FUNCTION "GCS7_BinCtrlSub" : VOID	// FC 67
TITLE = Bin Control: Subroutines
//COPYRIGHT:    (C) 1994 BY  BUHLER LTD.
//                           CH-9240 UZWIL  SWITZERLAND
//
//PRODUCT:      GCS7
//
//TITLE:        BIN CONTROL: SUBROUTINS
//
//-------------------------------------------------------------------------
//
//IDENT:        AUTOR:              DEPT:                         DATE:
//FC67.2.8      A.Egli              CT3                           18-Mai-2006
//                WinAC is not compatible
//FC67.2.7      A.Egli              CT3                           07-Jul-2004
//              DPFault per bin
//FC67.2.6      A.Egli              CT3                           08-Mar-2004
//              Per Bin bit InfIsInRecipe
//FC67.2.5      K.Tischer           CT3                           24-Oct-2003
//              - correction for StaLastBinActiv
//              - init test recipe 
//FC67.2.4      A.Egli              CT3                           04-Sep-2003
//              - check wit target value
//FC67.2.3      K.Tischer           CT3                           04-Jul-2003
//              - init DBW36 for decode
//FC67.2.2      A.Egli              CT3                           23-Jun-2003
//              - Set "BinDB".ToASW.BinActual also for Blend
//FC67.2.1      A.Egli              CT3                           05-Jun-2003
//              - Delete WeightTarget not before bin is deselected
//FC67.2.0      A.Egli              CT3                           07-Oct-2002
//              - New release 
//              - LastIngredient Active
//FC67.1.3      A.Egli              CT3                           06-Nov-01
//              subroutine 14: Init TestRefill
//FC67.1.2      A.Egli              AEE61                         14-Jan-98
//              Convert S5 to S7 (Version 1C)
//FC67.1.1      A.Egli              AEE61                         24-Jun-96
//              Convert S5 to S7 (Version 1C)
//
//-------------------------------------------------------------------------
//
//PURPOSE:      MANUAL : BINMAN
//
//RESTRICTIONS:
//
//-------------------------------------------------------------------------
//
//
//PARAMETER:
//------------
//  CODE: CODE OF CALLED FUNCTION
//        1  : Subroutine Test  Recipe
//        2  : Subroutine Read  Bin
//        3  : Subroutine Store Bin
//        4  : Subroutine Deselect All
//        5  : Subroutine Bin_Modify
//        6  : Subroutine Claer Value
//        7  : Subroutine Maske Active Bin
//        10 : Subroutine Read Ingredient
//        11 : Subroutine Read First Ingredient
//        12 : Subroutine Read Next Ingredient
//        13 : Subroutine Read_Blend_recipe
//
//ACTUAL DB BY CALL: DB Bin control
//AUFGESCHALGENER  : DB Siloverwaltung
//
//
AUTHOR : EA
FAMILY : GCS90UL
NAME : BIN_SUBR
VERSION : 2.8
VAR_INPUT
  CODE : INT ;	// CODE
END_VAR
VAR_TEMP
  BinNr : INT ;
  BinStatus : STRUCT
   InfLevelWarning : BOOL ;
   InfLevelFault1 : BOOL ;
   B10 : BOOL ;
   B11 : BOOL ;
   VarFlagOverwrite : BOOL ;
   InfLowLevel : BOOL ;
   InfLevelMiddle : BOOL ;
   InfHighLevel : BOOL ;
   InfActive : BOOL ;
   InfPreselect : BOOL ;
   InfDeselect : BOOL ;
   B3 : BOOL ;
   B4 : BOOL ;
   VarFlageLevelWarning : BOOL ;
   VarFlagLevelFault : BOOL ;
  END_STRUCT ;
  VarCntBin : INT ;
  VarAddrBin : DWORD ;
  VarCntIngr : INT ;
  VarAddrIngr : DINT ;
  VarBinNr : INT ;
  VarLenBinBit : INT ;	//Length of Bin data in bits
  VarLenIngrBit : INT ;	//Lenght per Ingr. in bits
  VarOkIngrCnt : INT ;	//Number of available ingredient (Transport)
  tmpNoTargetValue : BOOL ;
END_VAR
BEGIN
NETWORK
TITLE =
      L     DBW 10;	// "BinDB".Para.ParNoOfBytePerBin
      SLD   3;
      T     #VarLenBinBit;
      L     DBW 16;	// "BinDB".Para.ParNoOfBytePerIngr
      SLD   3;
      T     #VarLenIngrBit;
NETWORK
TITLE =  Subroutine Test Bin Status (Code=0)
//======================================
//
//Subroutine test bin Status: Code= 0
//-------------------------------------
//Input:
//Output:
//  DBX   43.0            // "BinDB".ToASW.InfActive
//  DBX   43.1            // "BinDB".ToASW.InfPreselect
//  DBX   43.2            // "BinDB".ToASW.InfDeselect 
//  DBX  103.0            // "BinDB".PCRead.Fault.EsLocked
//  DBX  103.1            // "BinDB".PCRead.Fault.EsLevelFault
//  DBX  105.7            // "BinDB".PCRead.Status.StaFeedOff
//  DBX   42.2            // "BinDB".ToASW.InfAllLocked
//  DBX   42.3            // "BinDB".ToASW.InfAllLevelFault
//
      L     #CODE;
      L     0;
      <>I;
      JC    aEnd;
      R     DBX 43.0;	// "BinDB".ToASW.InfActive
      R     DBX 43.1;	// "BinDB".ToASW.InfPreselect
      R     DBX 43.2;	// "BinDB".ToASW.InfDeselect 
      R     DBX 103.0;	// "BinDB".PCRead.Fault.EsLocked
      R     DBX 103.1;	// "BinDB".PCRead.Fault.EsLevelFault
      R     DBX 105.7;	// "BinDB".PCRead.Status.StaFeedOff
      R     DBX 104.3;	// "BinDB".PCRead.Status.StaDPFault     [2.7]
      S     DBX 42.2;	// "BinDB".ToASW.InfAllLocked
      S     DBX 42.3;	// "BinDB".ToASW.InfAllLevelFault
// [2.5] 
      S     DBX 43.4;	// "BinDB".ToASW.OutDryFillingDone
      L     0;
      T     DBW 56;	//"BinDB1".ToASW.OutActiveBinsCnt
      AN    DBX 7.0;	// ParObjectType=Blend
      JC    aAc1;
      T     DBW 48;	// "BinDB".ToASW.BinActual //[2.2]
//Start Adress Loop
aAc1: L     DBW 8;	//"BinDB".Para.ParByteFirstBin
      +     2;
      SLD   3;
      T     #VarAddrBin;	//--> Pointer to statusword of the bin
// (--loop bin: test  ----------)
      L     0;
      L     DBW 12;	//  "BinDB".Para.ParNoOfBin
      ==I;
      JC    aFER;
aLop: T     #VarCntBin;	// var_loop_bin_counter
      L     DBW [#VarAddrBin];	// binlist[n].Bin status word
      T     DBW 24;	//  )->var_bin_status
      AN    DBX 25.0;	//"BinDB".VarTemp.Bin.InfActiveBin
      JC    aEPY;
//Counter Active bins
      L     DBW 56;	//"BinDB1".ToASW.OutActiveBinsCnt
      +     1;
      T     DBW 56;	//"BinDB1".ToASW.OutActiveBinsCnt
      AN    DBX 7.0;	//[2.2 -->] ParObjectType=Blend
      JC    aAc2;
      L     #VarAddrBin;
      +     L#-16;
      LAR1;
      L     DBW [AR1,P#0.0];	// binlist[n].ParBinNr
      T     DBW 48;	// "BinDB".ToASW.BinActual     [<--2.2]
//Emptying Time
aAc2: LAR1  #VarAddrBin;
      L     DBW [AR1,P#2.0];	// binlist[n].ParEmptyingTime
      T     DBW 52;	// "BinDB".ToASW.OutEmptyingTimeBin
aEPY: A     DBX 25.0;	//"BinDB".VarTemp.Bin.InfActiveBin
      S     DBX 43.0;	// "BinDB".ToASW.InfActive
      A     DBX 25.1;	//"BinDB".VarTemp.Bin.InfPreselect
      S     DBX 43.1;	// "BinDB".ToASW.InfPreselect
      A     DBX 25.2;	// "BinDB".VarTemp.Bin.InfDeselect
      S     DBX 43.2;	//"BinDB".ToASW.InfDeselect
// --- DryFilling done ----------------
      A     DBX 25.0;	//"BinDB".VarTemp.Bin.InfActiveBin
      AN    DBX 24.3;	//"BinDB".VarTemp.Bin.OutDryFillingDone
      R     DBX 43.4;	// "BinDB".ToASW.OutDryFillingDone
// --- Feed Off ----------------
      A     DBX 25.0;	//"BinDB".VarTemp.Bin.InfActiveBin
      A     DBX 24.2;	//"BinDB".VarTemp.Bin.InFeedOff
      S     DBX 105.7;	// "BinDB".PCRead.Status.StaFeedOff
// --- DPFault ----------------
      A     DBX 25.0;	//"BinDB".VarTemp.Bin.InfActiveBin     [2.7]
      A     DBX 25.4;	//"BinDB".VarTemp.Bin.InOutDPFault     [2.7]
      S     DBX 104.3;	//"BinDB".PCRead.Status.StaDPFault     [2.7]
// --- Locked ----------------
      AN    DBX 24.0;	// bin[n]."BinDB".VarTemp.Bin.InfLocked
      JC    aR_W;
      A     DBX 25.0;	// "BinDB".VarTemp.Bin.InfActiveBin
      S     DBX 103.0;	// "BinDB".PCRead.Fault.EsLocked
      AN    DBX 25.6;	// "BinDB".VarTemp.Bin.VarFlagLocked
      S     DBX 25.6;	// "BinDB".VarTemp.Bin.VarFlagLocked
      S     DBX 41.0;	// "BinDB".ChangeBit.CBit1
      S     DBX 39.7;	// "BinDB".VarTemp.Value10.Flag7
      JU    aL_F;	// -- no warning --------------
aR_W: A     DBX 25.0;	// "BinDB".VarTemp.Bin.InfActiveBin
      R     DBX 42.2;	// "BinDB".ToASW.InfAllLocked
      A     DBX 25.6;	// "BinDB".VarTemp.Bin.VarFlagLocked
      R     DBX 25.6;	// "BinDB".VarTemp.Bin.VarFlagLocked 
      S     DBX 41.0;	// "BinDB".ChangeBit.CBit1
      S     DBX 39.7;	// "BinDB".VarTemp.Value10.Flag7
//---Faulted ----------------
aL_F: AN    DBX 24.1;	// "BinDB".VarTemp.Bin.InfLevelFault
      JC    aR_F;
//    --- fault ------------------
      A     DBX 25.0;	// "BinDB".VarTemp.Bin.InfActiveBin 
      S     DBX 103.1;	// "BinDB".PCRead.Fault.EsLevelFault
      AN    DBX 25.7;	// "BinDB".VarTemp.Bin.VarFlagLevelFault
      S     DBX 25.7;	// "BinDB".VarTemp.Bin.VarFlagLevelFault
      S     DBX 41.0;	// "BinDB".ChangeBit.CBit1 
      S     DBX 39.7;	// "BinDB".VarTemp.Value10.Flag7
      JU    aSAV;
//    -- no fault   --------------
aR_F: A     DBX 25.0;	//  "BinDB".VarTemp.Bin.InfActiveBin
      R     DBX 42.3;	//  "BinDB".ToASW.InfAllLevelFault 
      A     DBX 25.7;	//  "BinDB".VarTemp.Bin.VarFlagLevelFault
      R     DBX 25.7;	//  "BinDB".VarTemp.Bin.VarFlagLevelFault 
      S     DBX 41.0;	//  "BinDB".ChangeBit.CBit1 
      S     DBX 39.7;	// "BinDB".VarTemp.Value10.Flag7
//Store Bin
aSAV: L     DBW 24;	//   var_bin_status
      T     DBW [#VarAddrBin];	//   -> binlist[n].bin_status
      L     #VarAddrBin;
      L     #VarLenBinBit;
      +D;
      T     #VarAddrBin;	//   
      L     #VarCntBin;	//   
      LOOP  aLop;
//  (--END LOOP TEST -----------)
aFER: AN    DBX 43.0;	// "BinDB".ToASW.InfActive
      R     DBX 42.2;	// "BinDB".ToASW.InfAllLocked 
      R     DBX 42.3;	// "BinDB".ToASW.InfAllLevelFault 
      BEU;
aEnd: NOP   0;
NETWORK
TITLE = subroutine:Test recipe (Code 1)
//Input: DBW20="BinDB".VarTemp.InValue     = Source Recipe DBNr
//Input: DBW22="BinDB".VarTemp.BinNrByteNr = Source Recipe First Byte
//Output: DBW24=out.err_bin / BinStatus
//Output: DBW26=Number availabel ingredient 
//Output: DBW36=var_bin-number ingredient(error)
//Output: DBX39.1="BinDB".VarTemp.Value10.tmpLevelFault
//Output: DBX39.2="BinDB".VarTemp.Value10.tmpBinNotFound2
//Output: DBX39.3="BinDB".VarTemp.Value10.tmpEmptyRecipe
//Output: DBX39.4="BinDB".VarTemp.Value10.tmpFull
//Output: DBX39.6="BinDB".VarTemp.Value10.tmpLocked
//
      L     #CODE;
      L     1;
      <>I;
      JC    bEnd;
      S     DBX 39.6;	//"BinDB".VarTemp.Value10.tmpLocked
      S     DBX 39.1;	//"BinDB".VarTemp.Value10.tmpLevelFault
      S     DBX 39.4;	//"BinDB".VarTemp.Value10.tmpFull
      R     DBX 39.2;	//"BinDB".VarTemp.Value10.tmpBinNotFound2
      S     DBX 39.3;	//"BinDB".VarTemp.Value10.tmpEmptyRecipe
      L     0;	// [2.0]
      T     #VarOkIngrCnt;	// [2.0]
      T     DBW 36;	// [2.3]
// Init
      OPN   DI [DBW 20];	// Call Source DB: DBW20=inp.DB-Nr_source_recipe
      L     DBW 22;	// inp.ByteNrSourceRecipe
      +     6;	// Offset first ingredient
      SLD   3;	//   
      T     #VarAddrIngr;	//--> Address first ingredient
// ====START LOOP INGREDIENT =====
      L     0;
      L     DBW 18;	//  "BinDB".Para.ParNoOfIngr
      ==I;
      BEC;
bLoI: T     #VarCntIngr;
      L     DIW [#VarAddrIngr];	// load Ingredient bin number
      T     #VarBinNr;	// 
      L     0;	// 
      ==I;	// empty ingredient
      JC    bNXT;	// 
      L     DBW 8;	// "BinDB".Para.ParByteFirstBin
      SLD   3;	// 
      T     #VarAddrBin;	//--> Address of first bin
// ====START LOOP BIN ============
      L     1;
bLoB: T     #VarCntBin;	//   
      L     DBW 12;	// "BinDB".Para.ParNoOfBin 
      >I;
      JC    bErr;
      L     DBW [#VarAddrBin];	// load bin-number from bin list
      L     #VarBinNr;	// 
      ==I;	//  
      JC    bLEV;	//  
      L     #VarAddrBin;	//  
      L     #VarLenBinBit;	//  
      +D;	//  
      T     #VarAddrBin;	//  --> Address of bin
      L     #VarCntBin;	//  
      +     1;
      JU    bLoB;
// ====END LOOP BIN ==============
bLEV: L     DBD [#VarAddrBin];	// load bin[n].BinNr / BinStatus
      T     DBW 24;	// 
      L     1;
      L     #VarCntIngr;	//  
      ==I;	// --> (last loop ==special bin)
      AN    DBX 7.0;	// ParObjectType=Blend
      JC    bNXT;	// 
      AN    DBX 24.0;	// "BinDB".VarTemp.Bin.InfLocked 
      R     DBX 39.6;	// "BinDB".VarTemp.Value10.tmpLocked
      AN    DBX 24.1;	// "BinDB".VarTemp.Bin.InfLevelFault
      R     DBX 39.1;	// "BinDB".VarTemp.Value10.tmpLevelFault  
      A     DBX 39.3;	// "BinDB".VarTemp.Value10.tmpEmptyRecipe
      R     DBX 39.3;	// "BinDB".VarTemp.Value10.tmpEmptyRecipe
      AN    DBX 24.1;	// "BinDB".VarTemp.Bin.InfLevelFault  
      AN    DBX 24.6;	// "BinDB".VarTemp.Bin.InfLevelMiddle 
      AN    DBX 24.7;	// "BinDB".VarTemp.Bin.InfHighLevel  
      R     DBX 39.4;	// "BinDB".VarTemp.Value10.tmpFull  
      A     DBX 24.0;	// "BinDB".VarTemp.Bin.InfLocked     [2.0]
      O     DBX 24.1;	// "BinDB".VarTemp.Bin.InfLevelFault [2.0]
      JC    bNXT;	//                                   [2.0]
      L     #VarOkIngrCnt;	//                                   [2.0]
      +     1;	//                                   [2.0]
      T     #VarOkIngrCnt;	//                                   [2.0]
bNXT: L     #VarAddrIngr;	// 
      L     #VarLenIngrBit;	//   
      +D;	// 
      T     #VarAddrIngr;	// --> address next ingredient
      L     #VarCntIngr;	//   
      LOOP  bLoI;
      L     0;
      T     DBW 24;	//-> out.err_bin
      L     #VarOkIngrCnt;	//                                   [2.0]
      T     DBW 26;	//-->Number availabel ingredient     [2.0]
// ====END LOOP INGREDIENT =======
      BEU;
bErr: L     #VarBinNr;	//  var_bin-number ingredient
      T     DBW 36;	//  ->VarTemp.Value9                        
      S     DBX 39.2;	//  "BinDB".VarTemp.Value10.tmpBinNotFound2
      L     #VarOkIngrCnt;	//                                   [2.5]
      T     DBW 26;	//-->Number availabel ingredient     [2.5]
      BEU;
bEnd: NOP   0;
NETWORK
TITLE =  subroutine: Read bin (Code=2)
      L     #CODE;
      L     2;
      <>I;
      JC    cEnd;
      R     DBX 39.0;	// "BinDB".VarTemp.Value10.tmpBinNotFound1
      L     DBW 8;	// "BinDB".Para.ParByteFirstBin
      SLD   3;
      T     #VarAddrBin;
// ====START LOOP BIN ============
      L     1;
cLoB: T     #VarCntBin;	//   
      L     DBW 12;	// "BinDB".Para.ParNoOfBin
      >I;	// 
      JC    cErr;	// --> err: bin_not_found
      L     DBW [#VarAddrBin];	// load bin-number from bin list
      L     DBW 20;	// "BinDB".VarTemp.InValue= var_bin-number
      ==I;
      JC    cREA;
      L     #VarAddrBin;
      L     #VarLenBinBit;
      +D;
      T     #VarAddrBin;	// --> Address next bin
      L     #VarCntBin;
      +     1;
      JU    cLoB;
// ====END LOOP BIN ==============
cREA: L     #VarAddrBin;
      LAR1;
      SRD   3;
      T     DBW 22;	// Byte Nr of actual Bin
      L     DBD [AR1,P#2.0];
      T     DBD 24;	// -->"BinDB".VarTemp.StatusWord /"BinDB".VarTemp.ParEmpytingTime
      L     DBD [AR1,P#6.0];
      T     DBD 28;	// -->"BinDB".VarTemp.Bin.WeightActual
      L     DBW 10;	// "BinDB".Para.ParNoOfBytePerBin
      L     14;
      <I;
      BEC;	// If with target value
      L     DBD [AR1,P#10.0];
      T     DBD 32;	// -->"BinDB".VarTemp.Bin.WeightTarget
      BEU;
// ==== bin ot found ==============
cErr: S     DBX 39.0;	//  "BinDB".VarTemp.Value10.tmpBinNotFound1 
//      L     DBW   20                    // "BinDB".VarTemp.InValue
//      T     DBW   96                    // )-->"BinDB".PCRead.ErrElement
//      L     30                          //  )  error:bin_not_found
//      T     DBW   98                    //  )-> "BinDB".PCRead.ErrCode
      BEU;
cEnd: NOP   0;
NETWORK
TITLE =  subroutine: Store bin
      L     #CODE;	// )
      L     3;	// )  CODE= KF+3
      <>I;	// )
      JC    dEnd;	// )
      A     DBX 39.0;	// "BinDB".VarTemp.Value10.tmpBinNotFound1
      BEC;	//  )
      L     DBW 22;	//  ) Byte Number actual bin
      SLD   3;	//--> VarAddrBin
      LAR1;
      L     DBW [AR1,P#0.0];	// Actual bin
      L     DBW 20;	// var_bin-number
      <>I;	// 
      BEC;	// 
      L     DBW 24;	// var_bin_status
      T     DBW [AR1,P#2.0];	// -> bin[n].bin_status
      L     DBD 28;	//  "BinDB".VarTemp.Bin.WeightActual 
      T     DBD [AR1,P#6.0];	// -> bin[n].WeightActual
      L     DBW 10;	// "BinDB".Para.ParNoOfBytePerBin
      L     14;
      <I;
      BEC;
      L     DBD 32;	// "BinDB".VarTemp.Bin.WeightTarget
      T     DBD [AR1,P#10.0];	//  -> bin[n].WeightTarget
      BEU;
dEnd: NOP   0;
NETWORK
TITLE =  subroutine: Deselect all (Code=4)
      L     #CODE;
      L     4;
      <>I;
      JC    eEnd;
// === Deselect bin ==============
      L     DBW 8;	// "BinDB".Para.ParByteFirstBin
      SLD   3;
      LAR1;	//-->  Address bin
//  (--loop bin deselect --------)
      L     0;
      L     DBW 12;	// "BinDB".Para.ParNoOfBin  
      ==I;
      BEC;
eLOP: T     #VarCntBin;
      A     DBX [AR1,P#3.0];	// Bin[x].InfActiveBin
      S     DBX [AR1,P#3.2];	// Bin[x].InfDeselect
      SET;	// 
      R     DBX [AR1,P#3.1];	// Bin[x].InfPreselect
      TAR1;	// Address read
      L     #VarLenBinBit;	// 
      +D;	// 
      LAR1;	// --> Address next bin
      L     #VarCntBin;
      LOOP  eLOP;
// ====END LOOP DESELECT BIN =====
      BEU;
eEnd: NOP   0;
NETWORK
TITLE =  subroutine: Bin Modify (Code=5)
      L     #CODE;
      L     5;
      <>I;
      JC    fEnd;
// === Deselect bin ==============
      L     DBW 8;	// "BinDB".Para.ParByteFirstBin 
      SLD   3;
      LAR1;	//-->  Address bin
      AN    DBX 63.1;	// "BinDB".ToSSW.CmdReadyForSelect
      A     DBX 43.1;	//  "BinDB".ToASW.InfPreselect
      A     DBX 63.2;	// "BinDB".ToSSW.CmdReadyForDeselect
      R     DBX 63.2;	// "BinDB".ToSSW.CmdReadyForDeselect  
      AN    DBX 63.1;	// "BinDB".ToSSW.CmdReadyForSelect
      A     DBX 43.1;	// "BinDB".ToASW.InfPreselect
      JC    fX2;	// 
      L     DBW 50;	// "BinDB".ToASW.BinPreselected
      T     DBW 48;	// "BinDB".ToASW.BinActual 
//(--loop bin deselect --------)
fX2:  L     0;	//  
      L     DBW 12;	//  "BinDB".Para.ParNoOfBin
      ==I;
      JC    fIni;
fLop: T     #VarCntBin;
      SET;	//[2.8] WinAC
      A     DBX 63.2;	//"BinDB".ToSSW.CmdReadyForDeselect
      A     DBX [AR1,P#3.2];	// binlist[x].InfDeselect
      R     DBX [AR1,P#3.0];	// binlist[x].InfActiveBin
      R     DBX [AR1,P#3.2];	// binlist[x].InfDeselect
      S     DBX 41.0;	// "BinDB".ChangeBit.CBit1
      S     DBX 43.3;	// "BinDB".ToASW.CmdNewWay
      A     DBX 63.1;	// "BinDB".ToSSW.CmdReadyForSelect 
      A     DBX [AR1,P#3.1];	// binlist[x].InfPreselect
      S     DBX [AR1,P#3.0];	// binlist[x].InfActiveBin
      R     DBX [AR1,P#3.1];	// binlist[x].InfPreselect
      S     DBX 41.0;	// "BinDB".ChangeBit.CBit1  
      S     DBX 43.3;	// "BinDB".ToASW.CmdNewWay
      TAR1;	// Address read
      L     #VarLenBinBit;	// 
      +D;	// 
      LAR1;	// --> Address next bin
      L     #VarCntBin;
      LOOP  fLop;
// ====END LOOP DESELECT BIN =====
fIni: SET;
      R     DBX 63.1;	// "BinDB".ToSSW.CmdReadyForSelect
      R     DBX 63.2;	// "BinDB".ToSSW.CmdReadyForDeselect
      BEU;
fEnd: NOP   0;
NETWORK
TITLE =  subroutine: Clear Value (Code=6)
      L     #CODE;
      L     6;
      <>I;
      JC    gEnd;
// === Deselect bin ==============
      L     #VarLenBinBit;	// 
      L     80;	// [2.4]
      <I;
      BEC;	//    == no actual value
      L     DBW 8;	// "BinDB".Para.ParByteFirstBin
      SLD   3;	// 
      LAR1;	//-->  Address bin
//  (--loop bin bin -------------)
      L     0;
      L     DBW 12;	//  "BinDB".Para.ParNoOfBin
      ==I;
      JC    gIni;
gLop: T     #VarCntBin;
      L     0;	// (Clear Value)
      T     DBD [AR1,P#6.0];	//  binlist[n].WeightActual
      TAR1;	// 
      L     #VarLenBinBit;	// 
      +D;	// 
      LAR1;	//--> Address next bin
      L     #VarCntBin;
      LOOP  gLop;
// ====END LOOP BIN =====
gIni: BEU;
gEnd: NOP   0;
NETWORK
TITLE =  subroutine: Read Ingredient (Code 10)
//DBW20: : BinNr Ingredient
      L     #CODE;
      L     10;
      <>I;
      JC    C11;
      R     DBX 39.0;	// "BinDB".VarTemp.Value10.tmpBinNotFound1 
      L     DBW 14;	// "BinDB".Para.ParByteRecipeMemory  
      +     6;	// Offset fisrt ingredient in recipe
      SLD   3;	// 
      T     #VarAddrIngr;	// ->Address recipe
      OPN   DI [DBW 4];	// DB[Bin.ParSecDB ]
// ====START LOOP INGREDIENT =====
      L     0;
iLop: T     DBW 54;	// "BinDB".ToASW.VarIngrCnt
      L     DBW 18;	// "BinDB".Para.ParNoOfIngr
      >=I;	// 
      JC    iErr;	// 
      +     -1;	// 
      >=I;	// 
      AN    DBX 105.2;	// "BinDB".PCRead.Status.StaSpecialBin
      JC    iErr;	// 
      L     DIW [#VarAddrIngr];	// load ingredient
      L     DBW 20;	// "BinDB".VarTemp.InValue = InBinNr
      ==I;	// 
      BEC;	// 
      L     #VarAddrIngr;	// Address recipe
      L     #VarLenIngrBit;	// par_nr_of_byte_per_ingredient
      +D;	// 
      T     #VarAddrIngr;	// ->Address recipe
      L     DBW 54;	// "BinDB".ToASW.VarIngrCnt
      +     1;	// 
      JU    iLop;
// ====END LOOP INGREDIENT =======
iErr: S     DBX 39.0;	// "BinDB".VarTemp.Value10.tmpBinNotFound1
      L     0;	// 
      T     DBW 54;	// "BinDB".ToASW.VarIngrCnt
      BEU;
NETWORK
TITLE =  subroutine: Read First/Next Ingr (Code 11, 12)
//DBW20: "BinDB".VarTemp.InValue = OutBinNr
C11:  L     #CODE;
      L     11;	// CODE= 11 (fisrt ingredient)
      <>I;
      JC    C12;
      L     0;
      T     DBW 54;	// "BinDB".ToASW.VarIngrCnt 
      JU    jN_I;
C12:  L     #CODE;
      L     12;	// CODE= 12 (Next ingredient)
      <>I;
      JC    C13;
      L     DBW 54;	// "BinDB".ToASW.VarIngrCnt
      +     1;	//  
      T     DBW 54;	// "BinDB".ToASW.VarIngrCnt
//Find
jN_I: R     DBX 39.0;	//  "BinDB".VarTemp.Value10.tmpBinNotFound1
      L     DBW 14;	//  "BinDB".Para.ParByteRecipeMemory
      +     6;	// Offset first ingedient in recipe
      SLD   3;	// 
      T     #VarAddrIngr;	// ->Address recipe
      OPN   DI [DBW 4];	// DB[Bin.Para.ParSecDB ]
      AN    DBX 105.2;	// "BinDB".PCRead.Status.StaSpecialBin
      JC    jOk;	// 
      L     DBW 54;	// "BinDB".ToASW.VarIngrCnt
      L     DBW 18;	// "BinDB".Para.ParNoOfIngr 
      +     -1;	// 
      >=I;	// 
      JC    jOk;	// 
      T     DBW 54;	// -->"BinDB".ToASW.VarIngrCnt 
jOk:  L     DBW 54;	// "BinDB".ToASW.VarIngrCnt 
      L     #VarLenIngrBit;
      *I;
      L     #VarAddrIngr;
      +D;
      T     #VarAddrIngr;
// ====START LOOP INGREDIENT =====
      L     DBW 54;
jLop: T     DBW 54;	// "BinDB".ToASW.VarIngrCnt
      L     DBW 18;	// "BinDB".Para.ParNoOfIngr 
      >=I;
      JC    jErr;
      +     -1;
      >=I;
      AN    DBX 105.2;	// "BinDB".PCRead.Status.StaSpecialBin 
      JC    jErr;
      L     DIW [#VarAddrIngr];	// load ingredient
      T     DBW 20;	// -> "BinDB".VarTemp.InValue = OutBinNr
      L     0;	//  no ingredient
      <>I;	//  
      BEC;	// -->found
//Next ingr
      L     #VarAddrIngr;	// 
      L     #VarLenIngrBit;	// ParNrOfBytePerIngredient
      +D;	// 
      T     #VarAddrIngr;	//  
      L     DBW 54;	// "BinDB".ToASW.VarIngrCnt
      +     1;	// 
      JU    jLop;
// ====END LOOP INGREDIENT =======
jErr: S     DBX 39.0;	// "BinDB".VarTemp.Value10.tmpBinNotFound1
      L     0;	// 
      T     DBW 54;	// "BinDB".ToASW.VarIngrCnt 
      BEU;
C13:  NOP   0;
NETWORK
TITLE =  subroutine: Read Blend Recipe (Code 13)
      L     #CODE;
      L     13;
      <>I;
      JC    C14;
      L     #VarLenBinBit;
      L     112;	//[2.4]
      <I;
      =     #tmpNoTargetValue;	//[2.6]
      SET;	//[2.6]
      R     DBX 39.0;	// "BinDB".VarTemp.Value10.tmpBinNotFound1
      S     DBX 39.3;	// "BinDB".VarTemp.Value10.tmpEmptyRecipe
      L     0;	//  
      L     DBW 12;	//"BinDB".Para.ParNoOfBin
      ==I;
      BEC;	// 
      OPN   DI [DBW 4];	// DB[Bin.Para.ParSecDB ]
      L     DBW 8;	//  "BinDB".Para.ParByteFirstBin 
      SLD   3;
      T     #VarAddrBin;
      LAR1;
      AN    DBX 21.1;	// VarTemp.InValue1= Code=read target Value
      JC    kSta;	// 
// -- Loop Clear ---
      L     DBW 12;	// par_nr_of_bin
kLoC: T     #VarCntBin;	// var_loop_bin_counter
      A     DBX [AR1,P#3.0];	// bin[n].InfActiveBin     [2.1]
      O     DBX [AR1,P#3.2];	// bin[n].InfDeselect      [2.1]
      O     #tmpNoTargetValue;	// [2.6]
      JC    kJ1;
      L     0;
      T     DBD [AR1,P#10.0];	// Bin[x].WeightTarget
kJ1:  R     DBX [AR1,P#3.5];	// bin[n].InfIsInRecipe    [2.6]
      L     #VarLenBinBit;
      +AR1;	// var_addr_bin
      L     #VarCntBin;	// var_loop_bin_counter
      LOOP  kLoC;
// -- End loop claer ---
kSta: L     DBW 14;	//  "BinDB".Para.ParByteRecipeMemory
      +     6;	// Offset First ingredient
      SLD   3;
      LAR2;	//->Address recipe ingredient
//  (--START LOOP INGREDIENT ----)
      L     1;
kLoI: T     #VarCntIngr;
      L     DBW 18;	// "BinDB".Para.ParNoOfIngr
      >I;
      BEC;
      L     DIW [AR2,P#0.0];	// load ingredient
      T     #VarBinNr;	// ->bin-number ingredient
      L     0;	// 
      ==I;	// empty ingredient
      JC    kNxI;	// 
      R     DBX 39.3;	//  "BinDB".VarTemp.Value10.tmpEmptyRecipe
// --START LOOP SEARCH BIN -----
      LAR1  #VarAddrBin;	//  
      L     DBW 12;	// par_nr_of_bin
kLoB: T     #VarCntBin;	// 
      L     DBW [AR1,P#0.0];	// load bin-number from bin list
      L     #VarBinNr;	// bin number ingredient
      ==I;
      JC    kON;
      TAR1;	// 
      L     #VarLenBinBit;	// nr_of_DW_per_bin
      +D;
      LAR1;	// address next bin in bin list
      L     #VarCntBin;
      LOOP  kLoB;
      JU    kErr;	// --> err: bin_not_found
// -- End loop search bin ----
kON:  S     DBX [AR1,P#3.5];	// bin[n].InfIsInRecipe    [2.6]
      AN    DBX 21.0;	// VatTemp.InValue=1: code=preselect
      JC    kF2;
      AN    DBX [AR1,P#3.0];	// bin[n].InfActiveBin
      S     DBX [AR1,P#3.1];	// bin[n].InfPreselect
      A     DBX [AR1,P#3.2];	// bin[n].InfDeselect
      R     DBX [AR1,P#3.2];	// bin[n].InfDeselect
kF2:  AN    DBX [AR1,P#3.0];	// bin[n].InfActiveBin
      AN    DBX 7.3;	// "BinDB".Para.ParTypeDef.ParWithTargetValue
      ON    DBX 21.1;	// code=target_value
      O     #tmpNoTargetValue;	// [2.6]
      JC    kNxI;
      L     DID [AR2,P#2.0];	// load_target value
      T     DBD [AR1,P#10.0];	//-> bin.target_value
kNxI: TAR2;
      L     #VarLenIngrBit;	// par_nr_of_DW_per_ingredient
      +D;
      LAR2;	//->Address next ingredient
      L     #VarCntIngr;
      +     1;
      JU    kLoI;
//===END LOOP INGREDIENT ======)
kErr: NOP   0;
//      L     #VarBinNr
//      T     DBW   96                    //-->"BinDB".PCRead.ErrElement
//      L     30                          // error:bin_not_found
//      T     DBW   98                    // ->"BinDB".PCRead.ErrCode
      S     DBX 39.0;	// "BinDB".VarTemp.Value10.tmpBinNotFound1
      BEU;
NETWORK
TITLE =  subroutine: Init TestRefill
//This routine is used by Scale Contro: Test Refill Level
C14:  L     #CODE;
      L     14;
      <>I;
      JC    rEnd;
      L     DBW 8;	// "BinDB".Para.ParByteFirstBin
      SLD   3;
      LAR1;	//-->  Address bin
//  (--loop bin deselect --------)
      L     0;
      L     DBW 12;	//  )  par_nr_of_bin
      ==I;
      BEC;
rLOP: T     #VarCntBin;
      SET;
      R     DBX [AR1,P#3.1];	// bin[n].InfPreselect
      R     DBX [AR1,P#2.6];	// bin[n].InfLevelMiddle
      TAR1;
      L     #VarLenBinBit;	// 
      +D;	// 
      LAR1;	// --> Address next bin
      L     #VarCntBin;	// var_loop_bin_counter
      LOOP  rLOP;
// ====END LOOP DESELECT BIN =====
      BEU;
rEnd: NOP   0;
NETWORK
TITLE =
END_FUNCTION

FUNCTION "GCS7_ScaleCtrlMain" : VOID	// FC 68
TITLE = Scale Control: Main routines
//COPYRIGHT:    (C) 1994 BY  BUHLER LTD.
//                           CH-9240 UZWIL  SWITZERLAND
//
//PRODUCT:      GCS7
//
//TITLE:        SCALE CONTROL: MAIN PROGRAM
//
//Revision: 10
//
//-------------------------------------------------------------------------
//
//IDENT:        AUTOR:              DEPT:                         DATE:
//
//FC68.3.3      A.Egli              CT3                           18-Sep-2003
//              LAR1 and not +AR1
//FC68.3.2      A.Egli              CT3                           28-Aug-2003
//              BEB replaced with SPB NEXT
//FC68.3.1      A.Egli              CT3                           14-Mar-2003
//              Line-DB ParScales[1..64] removed
//FC68.3.0      A.Egli              CT3                           07-Okt-2002
//              New release with 64 Scales
//FC68.2.0      A.Egli              CT3                           12-Mar-2000
//              Any offset in section DB: GCPROVB: Revision 2
//              Test Refill Level: Set InfLevelMiddle if LLevel is uncovered
//FC68.1.5      A.Egli              CT3                           12-Mar-2000
//              Replace DBW120 with DBD120
//FC68.1E       A.Egli              CT3                           11-Aug-99
//              PC Direct Control: Check commands
//              Release scale for dosing if scale not in recipe mode
//FC68.1D       A.Egli              CT3                           13-Aug-98
//              PC Direct Control DBB52 replace by DBD52
//FC68.1C       A.Egli              CT3                           24-Jun-98
//              Start only used scales
//FC68.1B       A.Egli              AEE61                         16-Jan-98
//              Update to S5 Version 2G
//
//FC68.1A       A.Egli              AEE61                         25-Sep-96
//              Convert from S5 Version 2F
//
//-------------------------------------------------------------------------
//
//PURPOSE:      MANUAL : SCMAN
//
//RESTRICTIONS:
//
//-------------------------------------------------------------------------
//
//FC-PARAMETER:
//------------
//  CODE: CODE DER AUSZUFUEHRENDEN FUNKTION    Format: D    examp. KF+ 1
//        KF +0    : METHODE CONTROL-SECTION
//        KF +1    : METHODE DECODER
//        KF +2    : METHODE INIT DATA
//        KF +7    : METHODE O_SCALE
//        KF +8    : METHODE DIAGNOSE
//        KF +12   : METHODE TestRefillLevel
//
//
//
AUTHOR : EA
FAMILY : GCS7UL
NAME : SCC_MAN
VERSION : 3.3
VAR_INPUT
  CODE : INT ;	// CODE
  Sec : UDT 10680;
END_VAR
VAR_TEMP
  ParScaleInSection : ARRAY  [1 .. 2 ] OF //Must be at LD0
  DINT ;
  ToASW : STRUCT
   spare0 : BOOL ;
   EsRefillLevel : BOOL ;
   CmdTestRefillDone : BOOL ;
   spare3 : BOOL ;
   spare4 : BOOL ;
   spare5 : BOOL ;
   spare6 : BOOL ;
   spare7 : BOOL ;
   InfActive : BOOL ;
   InfEmptying : BOOL ;
   CmdReady : BOOL ;
   CmdEmptied : BOOL ;
   InfFault : BOOL ;
  END_STRUCT ;
  ToSSW : STRUCT
   InfEnableDosing : BOOL ;
   spare1 : BOOL ;
   spare2 : BOOL ;
   spare3 : BOOL ;
   spare4 : BOOL ;
   spare5 : BOOL ;
   spare6 : BOOL ;
   spare7 : BOOL ;
   CmdReset : BOOL ;
   CmdAbortBatch : BOOL ;
   CmdAcceptWt : BOOL ;
   CmdRetry : BOOL ;
  END_STRUCT ;
  CmdStartScales : ARRAY  [1 .. 2 ] OF //Must be at LD12
  DINT ;
  InfActiveScales : ARRAY  [1 .. 2 ] OF //Must be at LD20
  DINT ;
  InfEmptiedScales : ARRAY  [1 .. 2 ] OF //Must be at LD28
  DINT ;
  tmpFinalyDischarge : ARRAY  [1 .. 2 ] OF //Must be at LD36
  DINT ;
  tmpScaleUsed : ARRAY  [1 .. 2 ] OF //Must be at LD44
  DINT ;
  tmpFault : BOOL ;
  tmpScaleDB : INT ;
  tmpScaleNr : DINT ;
  tmpScaleIdx : INT ;
  tmpLineNr : INT ;
  tmpScaleBit : DINT ;
  tmpLineDB : INT ;
  tmpRecipePlace : INT ;
  tmpOffsetRecipe : INT ;
  tmpRecipeLen : INT ;
  tmpRecipeDB : INT ;
  tmpRecipeAddrSCDB : INT ;
  tmpRecipeAddrL_DB : INT ;
  tmpScalePara : BOOL ;
  tmpBinPara : BOOL ;
  tmpDBSource : INT ;
  tmpDWSource : INT ;
  tmpDBDestination : INT ;
  tmpDWDestination : INT ;
  tmpLenCopy : INT ;
  tmpDBPointer : DINT ;
  tmpSecDB : INT ;
  tmpInstanzDB : INT ;
  tmpInstanzPointer : DINT ;
  tmpBinDB : INT ;
  tmpBinControlDB : INT ;
END_VAR
BEGIN
NETWORK
TITLE =
      L     P##Sec;
      LAR1;
      L     W [AR1,P#0.0];
      T     #tmpInstanzDB;
      L     D [AR1,P#2.0];
      T     #tmpInstanzPointer;
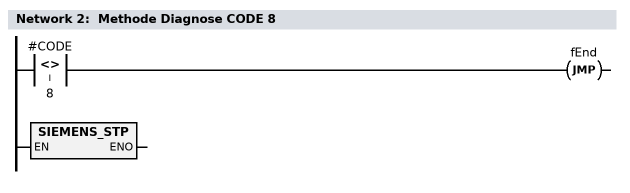
NETWORK
TITLE =  Methode Diagnose CODE 8
//ACTUAL DB BY CALL: not used
      L     #CODE;
      L     8;
      <>I;
      JC    fEnd;
//!!!!!!!!!!!!!!!!!!!!!!!!!!!!!!!!!!!!!!!!!!!!!!!!!!!!!!!!!
//Illegal function: This function is now part of the FC41
//                  Remove call FC68.Code=8
      CALL  "SIEMENS_STP";
//!!!!!!!!!!!!!!!!!!!!!!!!!!!!!!!!!!!!!!!!!!!!!!!!!!!!!!!!!
fEnd: NOP   0;
NETWORK
TITLE =  METHODE DECODER : Code 1
//ACTUAL DB BY CALL: Line DB
      L     #CODE;
      L     1;
      <>I;
      JC    dEnd;
      AN    DBX 145.0;	// "LineDB".JobWrite.Hsk.F_Define
      AN    DBX 145.1;	// "LineDB".JobWrite.Hsk.F_Execute
      AN    DBX 145.2;	// "LineDB".JobWrite.Hsk.F_Modify
      BEC;
      L     DBNO;
      T     #tmpLineDB;
      L     2#1;	// Mode=Copare with Job in L-DB
      T     DBW 22;	// "LineDB".VarTemp[2]= var_mode
//--- SUBROUTINE SEARCH_SECTION ---------
      CALL  "GCS7_SecCtrlSub" (
           CODE                     := 4);
      L     0;
      L     DBW 22;	//  "LineDB".VarTemp[2]  =OutSectionDB
      ==I;
      JC    dINI;
      T     #tmpSecDB;	// )->Target SectionDB
      OPN   DI [#tmpSecDB];	// >>>CALL Section_DB
      L     DIW 230;	// "SecDB".JobAc.RecipePlace
      A     DIX 200.7;	// "SecDB".JobAc.StaBatch.StaScaleRecipeValid
      T     #tmpRecipePlace;
      JC    dMOV;	// 
      T     DBW 20;	// ->L_DB.VarStartRecipePlace
      A     DBX 145.2;	// "LineDB".JobWrite.Hsk.F_Modify
      JC    dINI;	// 
//----Search recipe place-------------- 
//    SUBROUTINE SEARCH_RECIPE_PLAC
      CALL  "GCS7_ScaleCtrlSub" (
           CODE                     := 0);
      L     0;	//  
      L     DBW 20;	//  L_DB.VarRecipePlace
      >I;	//  
      JC    dER3;	//  
//----End Search recipe place ------------- 
      T     #tmpRecipePlace;
      OPN   DI [#tmpSecDB];	// >>>CALL section-DB
      T     DIW 230;	// ->"SecDB".JobAc.RecipePlace
      SET;	// 
      S     DIX 200.7;	// ->"SecDB".JobAc.StaBatch.StaScaleRecipeValid
dMOV: AN    DBX 145.2;	// "LineDB".JobWrite.Hsk.F_Modify 
      JC    dCOP;
//--- IF Modify: Test Scale dosing ---------- 
      L     1;
dLPS: T     #tmpScaleNr;	//  
      +     -1;
      LAR1;	//[3.3]
      AN    DBX [AR1,P#146.0];	// "LineDB".JobWrite.ObjMask[x]
      JC    dNXS;
      OPN   DI 8;
      L     #tmpScaleNr;
      T     DIW 20;	//--> DB8.ScaleNr
      CALL  "GCS7_ScaleCtrlSub" (
           CODE                     := 3);	// Subroutine ScalePointer
      L     DIW 22;	//<--DB8.ScaleDB
      T     #tmpScaleDB;
      L     0;	// No Scale
      ==I;
      JC    dNXS;
      L     DBW 2;	// L_DB.ParLineNr
      OPN   DI [#tmpScaleDB];
      L     DIW 266;	// SCDB.lineNr
      ==I;	// 
      A(;
      L     DBD 160;	//  "LineDB".JobNom.JobNr
      L     DID 258;	// SCDB.job-number
      ==D;	// 
      );
      A     DIX 43.7;	// SCDB.ScaleActive
      JC    dER2;	// 
dNXS: NOP   0;
      L     64;
      L     #tmpScaleNr;
      +     1;	// )
      >I;	// )
      JC    dLPS;
      JU    dCOP;
//--- End Test Modify -------------------
//=== Copy data to Scale DB =============
dCOP: L     1;
dLop: T     #tmpScaleNr;
      +     -1;
      T     #tmpScaleIdx;
//----Soubroutine Scale-DB
      OPN   DI 8;
      L     #tmpScaleNr;
      T     DIW 20;	//--> DB8.ScaleNr
      CALL  "GCS7_ScaleCtrlSub" (
           CODE                     := 3);	// Subroutine ScalePointer
      L     DIW 22;	//<--DB8.ScaleDB
      T     #tmpScaleDB;
      L     0;	// No Scale
      ==I;
      JC    dNxt;
//----Line.Subroutine BlockAdr
      L     #tmpScaleNr;
      T     DBW 20;	//-> "LineDB".VarTemp[1]= InObjNr
      CALL  "GCS7_LineCtrlSub" (
           CODE                     := 1);
      L     DBW 22;	// L_DB.VarDWNr
      T     #tmpRecipeAddrL_DB;
      L     0;	// 
      ==I;	// (not datablock for scale)
      JC    dNxt;
//----Soubroutine Recipe_pointer
      OPN   DI [#tmpScaleDB];	// >>> CALL Scale-DB
      L     DIW 104;	// REC .ParNrOfIngrPerRecipe
      L     DIW 106;	// SCDB.ParNrOfBytePerIngr
      *I;	// 
      T     #tmpRecipeLen;
      L     #tmpRecipePlace;
      *I;	// 
      L     DIW 100;	// REC.ParDwNrFirstRecipe
      +I;	// 
      T     #tmpRecipeAddrSCDB;
      L     DIW 98;	// REC.ParDBNrRecipe
      T     #tmpRecipeDB;
// -------------------------------
      OPN   DI 8;	// >>> DB8
      L     #tmpScaleDB;
      T     DIW 20;	// --> DB8.ScaleDB
      L     #tmpLineDB;
      T     DIW 22;	// -->DB8.VarSourceDB
      L     #tmpRecipeAddrL_DB;
      T     DIW 24;	// -->DB8.VarDWSource
//----Soubroutine Test_recipe---
      SET;
      R     DIX 27.0;	// -->DB8.TestSingleIngr.
      CALL  "GCS7_ScaleCtrlSub" (
           CODE                     := 2);
      A     DIX 39.0;	// <-FB69.DB8.fault
      JCN   dOk;
      L     DIW 26;	// <-FB69.DB8.error_bin
      T     DBW 138;	// -->"LineDB".JobRead.ErrElement
      L     DIW 28;	// <-FB69.DB8.error_code
      JU    dERO;
dOk:  CALL  "SYS_Copy_DBtoDB" (
           DBSource                 := #tmpLineDB,
           ByteSource               := #tmpRecipeAddrL_DB,
           DBDest                   := #tmpRecipeDB,
           ByteDest                 := #tmpRecipeAddrSCDB,
           NoOfByte                 := #tmpRecipeLen,
           Fault                    := #tmpFault);
      A     #tmpFault;
      JC    dER1;
      L     #tmpScaleIdx;
      LAR1;
      R     DBX [AR1,P#146.0];	// "LineDB".JobWrite.ObjMask[x]
dNxt: L     64;
      L     #tmpScaleNr;
      +     1;
      >I;
      JC    dLop;
// -- END LOOP SCALE -----------
dINI: BEU;
//=== ErrCode ======================
      L     20;	// err_code:illige objects
      JU    dERO;
dER3: L     40;	// err_code:no_recipe_memory
      JU    dERO;
dER2: L     #tmpScaleNr;
      T     DBW 20;	// L_DB.var_scale_nr
      L     43;	// err_code:no_read_recipe_mod
      JU    dERO;
dER1: L     42;	// err_code:cfg_fault_scale
dERO: T     DBW 140;	//-> "LineDB".JobRead.ErrCode 
      L     DBW 20;	//    L_DB.Scale-Nr
      T     DBW 142;	//-> "LineDB".JobRead.ErrObject
      BEU;
dEnd: NOP   0;
NETWORK
TITLE =  METHODE Init_Data: CODE:2
//ACTUAL DB BY CALL: Section-DB
//
      L     #CODE;
      L     2;
      <>I;
      JC    eEnd;
      LAR1  #tmpInstanzPointer;
      L     0;
      T     DBD [AR1,P#8.0];	// S_DB.ToASW/ToSSW
      T     DBD [AR1,P#12.0];	// S_DB.CmdStartScales
      T     DBD [AR1,P#20.0];	// S_DB.InfActiveScales[1]
      T     DBD [AR1,P#24.0];	// S_DB.InfActiveScales[2]
      T     DBD [AR1,P#28.0];	// S_DB.InfEmptiedScales[1]
      T     DBD [AR1,P#32.0];	// S_DB.InfEmptiedScales[2]
      BEU;
eEnd: NOP   0;
NETWORK
TITLE =  Copy to Stack: Code 0,12
//--Copy to temporare memory
      LAR1  #tmpInstanzPointer;
      L     DBD [AR1,P#0.0];
      T     #ParScaleInSection[1];
      L     DBD [AR1,P#4.0];
      T     #ParScaleInSection[2];
      L     DBD [AR1,P#8.0];
      T     LD 8;	//-->ToASW
      L     DBD [AR1,P#12.0];
      T     #CmdStartScales[1];
      L     DBD [AR1,P#16.0];
      T     #CmdStartScales[2];
      L     DBD [AR1,P#20.0];
      T     #InfActiveScales[1];
      L     DBD [AR1,P#24.0];
      T     #InfActiveScales[2];
      L     DBD [AR1,P#28.0];
      T     #InfEmptiedScales[1];
      L     DBD [AR1,P#32.0];
      T     #InfEmptiedScales[2];
NETWORK
TITLE =  METHODE CONTROL SECTION: CODE  0
//ACTUAL DB BY CALL: Section-DB
      L     #CODE;
      L     0;
      <>I;
      JC    aEND;
      R     #ToASW.InfEmptying;	//[3.2]  (this line moved)
      R     #ToASW.InfFault;	//[3.2]  (this line moved)
      A     #ToSSW.CmdRetry;
      R     #ToASW.EsRefillLevel;
//--Test active Scale -------- 
      L     0;	// )
      T     #tmpFinalyDischarge[1];
      T     #tmpFinalyDischarge[2];
      T     DBD 32;	// )   output total weigth registr.
      OPN   DI [DBW 4];	// >>> "SecDB".Para.ParLineDB
      L     DIW 2;	// "LineDB".Para.ParLineNr
      T     #tmpLineNr;
      L     1;
bLOP: T     #tmpScaleNr;
      +     -1;
      T     #tmpScaleBit;
      L     #tmpScaleNr;
      T     "GCS7_ScaleControlDB".VarTemp[1];	//--> DB8.ScaleNr
      CALL  "GCS7_ScaleCtrlSub" (
           CODE                     := 3);	// Subroutine ScalePointer
      L     "GCS7_ScaleControlDB".VarTemp[2];	//<--DB8.ScaleDB
      T     #tmpScaleDB;
      LAR1  #tmpScaleBit;
      OPN   DB [#tmpInstanzDB];
      AN    L [AR1,P#0.0];	// ParScaleInSection[x]
      JC    bDon;
      OPN   DI [#tmpScaleDB];	// >>> CALL scale-DB
      AN    DIX 42.5;	// SCDB.outp_readyForDischarge
      AN    DIX 232.1;	// Handshake.SendResult
      R     DIX 80.0;	// --> SCDB.FlagRegistation
      AN    DIX 249.0;	//StaRecipeAc [1D]
      A     DIX 253.0;	//StaSingleIngrMode [1D]
      S     DIX 54.2;	// ->SCDB.cmd_EnableDosingSec [1D]
      AN    DIX 55.0;	// CmdStartRecipe
      AN    DIX 249.0;	// StaRecipeAc
      JC    bDon;
      L     DBD 160;	// "SecDB".JobNom.JobNr
      L     DID 258;	// Scale.JobNumber
      <>D;	// 
      JC    bDon;
      L     DBW 206;	// "SecDB".JobAc.BatchNo
      L     DIW 264;	// SCDB.BatchNr
      <>I;	// 
      JC    bDon;
      L     DIW 266;	// SCDB.LineNr
      L     #tmpLineNr;
      <>I;	// 
      JC    bDon;
//--- Active Scales -----------------------
      AN    DBX 119.3;	// "SecDB".PCRead.Status.StaOnline
      =     DIX 55.7;	// ->SCDB.InpOffline
      A     #ToSSW.CmdReset;
      S     DIX 59.6;	// ->SCDB.cmd_reset
      A     #ToSSW.CmdAbortBatch;
      S     DIX 58.1;	// ->SCDB.abortBatch
      A     #ToSSW.CmdAcceptWt;
      S     DIX 58.0;	// ->SCDB.cmd_acceptWt
      A     #ToSSW.CmdRetry;
      S     DIX 59.7;	// ->SCDB.retry
      A     #ToSSW.InfEnableDosing;
      =     DIX 54.2;	// ->SCDB.cmd_EnableDosingSec
      AN    DIX 42.5;	// )   SCDB.outp_readyForDischarge
      O     DIX 54.5;	// )   SCDB.inp_closed
      ON    DIX 251.2;	// )   SCDB.sta_DischargeFinal
      AN    DIX 232.1;	// )   Handshake.SendResult
      O     DIX 80.0;	// )   SCDB.flag_registation
      JC    FLAG;	// )
      S     DIX 80.0;	// --> SCDB.flag_registation
      L     DIW 30;	// )   par_NrOfDecPoint
      L     0;	// )
      ==I;	// )
      L     1000;	// )   units
      JC    REG;	// )
      L     DIW 30;	// )   par_NrOfDecPoint
      L     1;	// )
      ==I;	// )
      L     100;	// )   units
      JC    REG;	// )
      L     DIW 30;	// )   par_NrOfDecPoint
      L     2;	// )
      ==I;	// )
      L     10;	// )   units
      JC    REG;	// )
      L     1;	// )   units
      JU    REG;
REG:  DTR;
      L     DID 278;	// )   SCDB.TotalWtActual
      DTR;	// )
      *R;	// )
      RND;
      L     DBD 32;	// )   output total weigth
      +D;	// )
      T     DBD 32;	// --> output total weigth
FLAG: A     DIX 42.5;	// SCDB.outp_readyForDischarge
      S     #ToASW.InfEmptying;
      A     DIX 43.4;	// SCDB.InfFault
      S     #ToASW.InfFault;
      LAR1  #tmpScaleBit;
      SET;
      S     L [AR1,P#20.0];	// InfActiveActive[x]
      A     DIX 251.2;	// SCDB.StaFinalDischarge
      LAR1  #tmpScaleBit;
      S     L [AR1,P#36.0];	// Out.tmpFinalDischarge[x]
      JU    bNXT;
bDon: LAR1  #tmpScaleBit;
      A     L [AR1,P#20.0];	// InfActiveScale[x]
      R     L [AR1,P#20.0];	// InfActiveScale[x]
      S     L [AR1,P#28.0];	// InfEmptiedScale[x]
bNXT: L     64;
      L     #tmpScaleNr;
      +     1;
      >I;
      JC    bLOP;
//======End Test active Scale ========== 
      A(;
      L     DBD 170;	//"SecDB".JobNom.ScaleUsed[32..1]
      L     #ParScaleInSection[1];
      AD;
      T     #tmpScaleUsed[1];
      L     #InfEmptiedScales[1];
      ==D;
      );
      A(;
      L     DBD 174;	//"SecDB".JobNom.ScaleUsed[64..33]
      L     #ParScaleInSection[2];
      AD;
      T     #tmpScaleUsed[2];
      L     #InfEmptiedScales[2];
      ==D;
      );
      =     #ToASW.CmdEmptied;
      A(;
      L     #InfEmptiedScales[1];
      L     #tmpFinalyDischarge[1];
      OD;
      L     #tmpScaleUsed[1];
      ==D;
      );
      A(;
      L     #InfEmptiedScales[2];
      L     #tmpFinalyDischarge[2];
      OD;
      L     #tmpScaleUsed[2];
      ==D;
      );
      O     #ToASW.CmdEmptied;
      =     #ToASW.CmdReady;
      L     0;
      L     DBD 32;	// Input: Weight for registration
      <>D;
      JCN   b000;
      CALL  "GCS7_SecCtrlMain" (
           CODE                     := 10);	// Sec : Methode SEC.ResultBatch
b000: NOP   0;
//==== start scales =============
      AN    DBX 45.7;	// Sec.InfDataReady
      JC    TEST;	// 
      L     1;
bLo2: T     #tmpScaleNr;
      +     -1;
      T     #tmpScaleBit;
      LAR1  #tmpScaleBit;
      A     L [AR1,P#0.0];	// ParScaleInSection[x]
      A     L [AR1,P#12.0];	// CmdStartScale[x]
      A     L [AR1,P#44.0];	// tmpScaleUsed[x]
      AN    L [AR1,P#28.0];	// InfEmptiedScale[x]
      AN    L [AR1,P#20.0];	// InfActiveScale[x]
      JCN   NEXT;	// 
//--- Start Scale --------
      OPN   DI 8;
      L     #tmpScaleNr;	// scale-nr
      T     DIW 20;	//--> DB8.ScaleNr
      CALL  "GCS7_ScaleCtrlSub" (
           CODE                     := 3);	// Subroutine ScalePointer
      L     DIW 22;	//<--DB8.ScaleDB
      T     #tmpScaleDB;
      OPN   DI [#tmpScaleDB];	// >>> call scale-DB
      AN    DIX 43.0;	//  SCDB.Inf_RecipeReq
      O     DIX 55.0;	//  SCDB.Cmd_StartRecipe
      JC    NEXT;	//[3.2]
      L     DBD 160;	// "SecDB".JobNom.JobNr
      T     DID 258;	// 
      L     DBW 178;	// "SecDB".JobNom.RecipeNr
      T     DIW 262;	// --> Scale.JobNumber
      L     DBW 206;	// "SecDB".JobAc.BatchNo
      T     DIW 264;	// --> Scale.BatchNr
      L     DBW 230;	// "SecDB".JobAc.RecipePlace
      T     DIW 70;	// --> Scale.Inf_RecipePlace
      L     DBW 218;	//  "SecDB".JobAc.BatchSizePpm
      T     DIW 268;	// --> Scale.BatchSizePc
      L     DBD 210;	// "SecDB".JobAc.BatchWeightTarget
      T     DID 270;	// --> Scale.BatchWtRecipe
      L     #tmpLineNr;
      T     DIW 266;	// --> Scale.LineNr
      SET;
      S     DIX 55.0;	// --> Scale.CmdStartRecipe
      LAR1  #tmpScaleBit;
      S     L [AR1,P#20.0];	// InfActiveActive[x]
//--- End Start Scale
NEXT: L     64;
      L     #tmpScaleNr;
      <=I;
      JC    TEST;
      +     1;
      JU    bLo2;
// ==== end loop scale ============
TEST: L     #InfActiveScales[1];
      L     0;
      <>D;
      O(;
      L     #InfActiveScales[2];
      L     0;
      <>D;
      );
      =     #ToASW.InfActive;
      L     0;
      T     #CmdStartScales[1];
      T     #CmdStartScales[2];
      SET;
      R     #ToSSW.CmdReset;
      R     #ToSSW.CmdAbortBatch;
      R     #ToSSW.CmdAcceptWt;
      R     #ToSSW.CmdRetry;
      JU    Save;
aEND: NOP   0;
NETWORK
TITLE =  Methode TestRefilLevel: Code 12
//ACTUAL DB BY CALL: Section-DB for testing
//Input:
//  S-DB: CmdTestRefillDone  : Flankenbit Meldung an PC erfolgt
//Output:
//  S-DB: EsRefillLevel      : Bin with level is found
//  S-DB: CmdTestRefillDone  : Flankenbit Meldung an PC erfolgt
//  S-DB: DBW 26             : BinNr with level-fault
      L     #CODE;
      L     12;
      <>I;
      JC    hEND;
      AN    #ToASW.EsRefillLevel;
      R     #ToASW.CmdTestRefillDone;
      SET;
      R     #ToASW.EsRefillLevel;
//======================================
//Init Bin Control
//[Rel 2.0 -->
      L     DBNO;
      T     #tmpSecDB;	// )->Target SectionDB
      L     1;	// 
//----LOOP:
hLo1: T     #tmpScaleNr;
      +     -1;
      LAR1;
      AN    DBX [AR1,P#170.0];	//"SecDB".JobNom.ScaleUsed[x]
      JC    hNx1;
      OPN   DI 8;
      L     #tmpScaleNr;	// )   scale-nr
      T     DIW 20;	//--> DB8.ScaleNr
      CALL  "GCS7_ScaleCtrlSub" (
           CODE                     := 3);	// Subroutine ScalePointer
      L     DIW 22;	//<--DB8.ScaleDB
      T     #tmpScaleDB;
      OPN   DI [#tmpScaleDB];
      L     DIW 32;	// CWA.ParDBBinControl
      T     #tmpBinControlDB;
      L     0;
      ==I;
      JC    hNx1;
      OPN   DB [#tmpBinControlDB];
      CALL  "GCS7_BinCtrlSub" (
           CODE                     := 14);	// Methode Init Test Refill
      OPN   DB [#tmpSecDB];
hNx1: L     64;
      L     #tmpScaleNr;	// S_DB.VarCntScale
      +     1;
      >=I;
      JC    hLo1;
//<--Rel 2.0]
//End Init Bin Control
//======================================
      L     1;	// 
//----LOOP:
hLop: T     #tmpScaleNr;
      +     -1;
      LAR1;
      OPN   DB [#tmpInstanzDB];
      AN    DBX [AR1,P#170.0];	// "SecDB".JobNom.ScaleUsed[x]
      JC    hNxt;
      L     #tmpScaleNr;
      T     "GCS7_ScaleControlDB".VarTemp[1];	//--> DB8.ScaleNr
      CALL  "GCS7_ScaleCtrlSub" (
           CODE                     := 3);	// Subroutine ScalePointer
      L     "GCS7_ScaleControlDB".VarTemp[2];	//<--DB8.ScaleDB
      T     #tmpScaleDB;
      T     "GCS7_ScaleControlDB".VarTemp[9];	// -> DB8.var_scale_DB_nr
      OPN   DB [#tmpInstanzDB];
      L     DBW 230;	//    Sec.InfRecipePlace
      T     "GCS7_ScaleControlDB".VarTemp[2];	// -> DB8.VarRecipePlace
// Subrotine TestLevel
      CALL  "GCS7_ScaleCtrlSub" (
           CODE                     := 5);
      L     "GCS7_ScaleControlDB".VarTemp[3];	//OutputFB69.VarDBBinControl
      T     #tmpBinDB;
      A     DB8.DBX 39.0;	// DB8.ErrorLevel
      JC    hErr;
hNxt: L     64;
      L     #tmpScaleNr;	// S_DB.VarCntScale
      +     1;
      >=I;
      JC    hLop;
      JU    Save;
hErr: L     "GCS7_ScaleControlDB".VarTemp[4];	// ErrBin
      OPN   DB [#tmpInstanzDB];
      T     DBW 26;	// SecDB.ErrBin
      S     #ToASW.EsRefillLevel;
      A     #ToASW.CmdTestRefillDone;
      O     DBX 102.0;	// "SecDB".PCRead.Hsk.F_Status
      JC    hNxt;
      S     DBX 102.0;	// "SecDB".PCRead.Hsk.F_Status
      S     DBX 41.0;	// "SecDB".ChangeBit.CBit1
      L     DBW 26;	// "SecDB".OutErrBin
      T     DBW 104;	// -> SecDB.PCRead.ErrElement
      L     48;	// Code=RefillLevel
      T     DBW 106;	// ->"SecDB".PCRead.ErrCode
      L     #tmpScaleNr;
      T     DBW 108;	// ->"SecDB".PCRead.ErrObject
      S     #ToASW.CmdTestRefillDone;
      JU    hNxt;
//      U     #ToASW.CmdTestRefillDone
//      AUF   DI [#tmpBinDB]              // >>> CALL DB Bin Control
//      O     DIX   94.0                  // "BinDB".PCRead.Hsk.F_Status
//      SPB   hNxt
//      S     DIX   94.0                  // "BinDB".PCRead.Hsk.F_Status
//      S     DIX  103.1                  // "BinDB".PCRead.Fault.EsLevelFault
//      S     DIX   41.0                  // "BinDB".ChangeBit.CBit1
//      L     DBD  160                    // "SecDB".JobNom.JobNr
//      T     DID  106                    // ->"BinDB".PCRead.JobNr
//      L     DBW  206                    // "SecDB".JobAc.BatchNo
//      T     DIW  110                    // "BinDB".PCRead.BatchNr
//      L     DBW   26                    // S_DB.OutErrBin
//      T     DIW   96                    // -> Bin.err_element
//      L     48                          // Code=RefillLevel
//      T     DIW   98                    // ->"BinDB".PCRead.ErrCode
//      S     #ToASW.CmdTestRefillDone
      JU    hNxt;
hEND: NOP   0;
NETWORK
TITLE =  Save:  Code 0,12
Save: NOP   0;
//--Copy to temporare memory
      OPN   DB [#tmpInstanzDB];
      LAR1  #tmpInstanzPointer;
      L     LD 8;	// ToASW
      T     DBD [AR1,P#8.0];	// S_DB.ToASW
      L     #CmdStartScales[1];
      T     DBD [AR1,P#12.0];
      L     #CmdStartScales[2];
      T     DBD [AR1,P#16.0];
      L     #InfActiveScales[1];
      T     DBD [AR1,P#20.0];
      L     #InfActiveScales[2];
      T     DBD [AR1,P#24.0];
      L     #InfEmptiedScales[1];
      T     DBD [AR1,P#28.0];
      L     #InfEmptiedScales[2];
      T     DBD [AR1,P#32.0];
NETWORK
TITLE =
END_FUNCTION

FUNCTION "GCS7_ScaleCtrlSub" : VOID	// FC 69
TITLE = Scale Control: Subroutines
//COPYRIGHT:    (C) 1994 BY  BUHLER LTD.
//                           CH-9240 UZWIL  SWITZERLAND
//
//PRODUCT:      GCS7
//
//TITLE:        SCALE CONTROL: SOUBROUTINS
//
//-------------------------------------------------------------------------
//
//IDENT:        AUTOR:              DEPT:                         DATE:
//
//FC69.2.0      A.Egli              CT3                           07-Okt-2002
//              New release with 64 Scales
//FC69.1.3      A.Egli              CT3                           06-Nov-01
//              Test Refill Level: Set bit InLevelMiddle,InPreselected
//
//FC69.1.2      A.Egli              AEE61                         21-Sep-98
//              Fault search recipe place
//
//FC69.1.1      A.Egli              AEE61                         25-Sep-96
//              Convert from S5 Version 1F
//
//-------------------------------------------------------------------------
//
//PURPOSE:      MANUAL : SCALEMAN
//
//RESTRICTIONS: only for 32-Bit CWA
//
//-------------------------------------------------------------------------
//
//
//FC-PARAMETER:
//------------
//  CODE: CODE OF CALLED FUNCTION
//        0  : Subroutine SearchFreeRecipePlace
//        2  : Subroutine Test Scale Recipe
//        3  : ScaleDB
//        5  : Test Level
//
//
//
AUTHOR : EA
FAMILY : GCSUL
NAME : SCC_SUB
VERSION : 2.0
VAR_INPUT
  CODE : INT ;	// CODE
END_VAR
VAR_TEMP
  tmpScaleDB : INT ;
  tmpScaleNr : DINT ;
  tmpBitAdr : DINT ;
  tmpRecipePlace : INT ;
  tmpBitNr : INT ;
  tmpUsedRecipe : DINT ;
  tmpNrOfIngr : INT ;
  tmpNrOfBitIngr : INT ;
  tmpNrOfBin : INT ;
  tmpNrOfBitBin : INT ;
  tmpCntBin : INT ;
  tmpCntIngr : INT ;
  tmpDBRecipe : INT ;
  tmpDBBin : INT ;
  tmpAddrIngr : DINT ;
  tmpAddrBin : DINT ;
  tmpBinControlDB : INT ;
  tmpBinNr : INT ;
END_VAR
BEGIN
NETWORK
TITLE =
NETWORK
TITLE = Subroutine ScaleDB: Code3
//ACTUAL DB BY CALL: not used
//
//Input:
//  DB8.DBW20 : ScaleNr
//Output:
//  DB8.DBW22 : ScaleDB
//
//======================================
//
//
      L     #CODE;
      L     3;
      <>I;
      JC    rEND;
      L     "GCS7_ScaleControlDB".VarTemp[1];	//Inp.ScaleNr
      SLD   4;
      LAR1;	//Bit-Nr.Pointer 
      L     DBW [AR1,P#40.0];
      T     "GCS7_ScaleControlDB".VarTemp[2];	//-->Out.ScaleDB
      BEU;
rEND: NOP   0;
NETWORK
TITLE =  Subroutine Search free recipe: Code 0
//ACTUAL DB BY CALL: Line-DB
//
//Input:
//  L_DB.DBW20: RecipePlace
//Output:
//  L_DB.DBW20: RecipePlace
//
      L     #CODE;
      L     0;
      <>I;
      JC    aEND;
      L     DBW 20;	//  input.recipe_place
      T     #tmpRecipePlace;
      L     0;
      T     #tmpUsedRecipe;
      OPN   DI [DBW 4];	// >>>CALL SECTION-DB DB["LineDB".Para.ParFirstSecDB]
aLOP: AN    DIX 45.7;	// "SecDB".ToASW.InfDataReady
      ON    DIX 200.7;	// "SecDB".JobAc.StaBatch.StaScaleRecipeValid
      JC    aNXT;	// 
      AN    DIX 44.7;	// "SecDB".ToASW.InfSameJobLineDB
      JC    aT2;	// 
      L     DIW 230;	// "SecDB".JobAc.RecipePlace
      T     #tmpRecipePlace;
aT2:  L     DIW 230;	// "SecDB".JobAc.RecipePlace
      L     DBW 10;	// "LineDB".Para.ParFirstRecipePlace
      -I;	// --> Bit-Nr.
      L     2#1;
      SLD;
      L     #tmpUsedRecipe;
      OD;
      T     #tmpUsedRecipe;
aNXT: L     0;
      L     DIW 8;	// "SecDB".Para.ParNextSecDB
      ==I;
      JC    aFID;
      OPN   DI [DIW 8];	// >>> CALL SECTION-DB  "SecDB".Para.ParNextSecDB]
      JU    aLOP;
// (--- End LOOP SECTION ------)
aFID: L     #tmpRecipePlace;
      T     DBW 20;	// InputRecipePlace
      L     DBW 10;	// "LineDB".Para.ParFirstRecipePlace
      <I;	// 
      JC    aNEW;
      -I;	// 
      T     #tmpBitNr;	// -->bit-number in mask
      L     DBW 8;	//  "LineDB".Para.ParNoOfRecipePlace
      >I;	// 
      JC    aNEW;	// 
      L     #tmpBitNr;
      L     #tmpUsedRecipe;
      SSD;
      SSD   1;	//   )
      JP    aNEW;	//   )->1=used
      BEC;	//   )
//----- Start loop find -----
aNEW: L     0;	// 
aLO2: T     #tmpRecipePlace;
      L     DBW 8;	// "LineDB".Para.ParNoOfRecipePlace
      >=I;	// 
      JC    aERO;	// ->no free recipe_place
      L     #tmpRecipePlace;	// RelRecipePlace
      L     #tmpUsedRecipe;
      SSD;
      SSD   1;	//   )
      JP    aNX2;	//   )->1=used
      L     #tmpRecipePlace;
      L     DBW 10;	// "LineDB".Para.ParFirstRecipePlace
      +I;	// 
      T     DBW 20;	// ->output.RecipePlace
      BEU;
aNX2: L     #tmpRecipePlace;
      +     1;	// 
      JU    aLO2;	// 
//---- End Loop find --------
aERO: L     -1;	// error_no free_recipe_place 
      T     DBW 20;
      BEU;
aEND: NOP   0;
NETWORK
TITLE =  Subroutine TestScaleRecipe Code 2
//ACTUAL DB BY CALL: not used
//Input:
//  DB8.DBW20   : ScaleDB
//  DB8.DBW22   : DB-Number source
//  DB8.DBW24   : DW-Number source
//  DB8.DBX27.0 : SingleIngrTest
//
//Output:
//  DB8.DW26  : err_bin
//  DB8.DBW28 : err_code
//  DB8.DBX39.0: err_fault
//
//
      L     #CODE;
      L     2;
      <>I;
      JC    bEND;
      R     DB8.DBX 39.0;	// ->output.fault
      L     "GCS7_ScaleControlDB".VarTemp[2];	// DB Source 
      T     #tmpDBRecipe;
      L     "GCS7_ScaleControlDB".VarTemp[3];	// ByteSource
      SLD   3;
      T     #tmpAddrIngr;
      L     "GCS7_ScaleControlDB".VarTemp[1];	// ScaleDB
      T     #tmpScaleDB;
      OPN   DI [#tmpScaleDB];	// >>> Call ScaleDB
      L     DIW 108;	// SCDB.ParDBBinData
      T     #tmpDBBin;
      L     DIW 110;	// SCDB.ParDWNrBinData
      SLD   3;
      T     #tmpAddrBin;
      L     DIB 105;	// ParNrOfIngrPerRecipe
      T     #tmpNrOfIngr;
      L     DIW 106;	// SCDB.ParNrOfByPerIngr
      SLD   3;
      T     #tmpNrOfBitIngr;
      L     DIB 113;	// ParNrOfBin
      T     #tmpNrOfBin;
      L     DIW 114;	// SCDB.ParNrOfByPerBin
      SLD   3;
      T     #tmpNrOfBitBin;
// --- Begin Loop ingredient ------
      L     0;
bLOI: T     #tmpCntIngr;
      L     #tmpNrOfIngr;
      >=I;
      JC    bOUT;
      OPN   DI [#tmpDBRecipe];	//  
      L     DIW [#tmpAddrIngr];	// Ingr[n].bin_nr
      T     #tmpBinNr;
      L     0;	// 
      ==I;	// -->end of recipe
      JC    bOUT;	// 
      <=I;	// Special bin
      JC    bNXI;	// 
      OPN   DI [#tmpDBBin];
      LAR1  #tmpAddrBin;
// ---Begin loop bin -----------
      L     0;
bLOB: T     #tmpCntBin;
      L     #tmpNrOfBin;
      >=I;	// 
      JC    bER0;	// => bin_not_found
      L     DIW [AR1,P#0.0];	// BinDB.bin[n].bin_nr
      L     #tmpBinNr;
      ==I;	// 
      JC    bNXI;	// -> next ingr.
      L     #tmpNrOfBitBin;
      +AR1;
      L     #tmpCntBin;	// -> var_bin_counter
      +     1;	// 
      JU    bLOB;	// 
//--- end loop bin ------------
bNXI: L     #tmpAddrIngr;
      L     #tmpNrOfBitIngr;
      +D;	// (increment read address)
      T     #tmpAddrIngr;
      A     DB8.DBX 27.0;	// test single ingr.
      JC    bOUT;	// ende
      L     #tmpCntIngr;
      +     1;
      JU    bLOI;
// --- end loop ingredient------
bER0: L     30;	// code: err_ingr_not_found
      JU    bERO;
      L     44;	// code: err_cfg_fault_bin_list
bERO: T     "GCS7_ScaleControlDB".VarTemp[5];	// ErrorCode
      S     DB8.DBX 39.0;	// --> output.fault
      L     #tmpBinNr;
      T     "GCS7_ScaleControlDB".VarTemp[4];	// var_bin_nr
      BEU;
bOUT: L     0;
      T     "GCS7_ScaleControlDB".VarTemp[5];	// --> error_code
      T     "GCS7_ScaleControlDB".VarTemp[4];	// var_bin_nr
      BEU;
bEND: NOP   0;
NETWORK
TITLE =  Subroutine TestLevel: Code 5
//ACTUAL DB BY CALL: not used
//Input:
//  DB8.DBW22  : tmpVar[2]  :=RecipePlace
//  DB8.DBW36  : tmpVar[9]  :=Scale-DB
//Output:
//  DB8.DBW26  : tmpVar[4]  :=err_bin
//  DB8.DBX39.0: tmpFault[8]:=OutFault
//               1= BinNotFound 
//  DB8.DBW24  : tmpVar[3]  :=par_DB-Nr_BinControl
//
      L     #CODE;	// )
      L     5;	// )  CODE= KF+5
      <>I;	// )
      JC    cEND;
      R     DB8.DBX 39.0;	// )->output.fault
      OPN   DI [DBW 36];	// >>> Call ScaleDB
      L     DIW 98;	// ParDBNrRecipe
      T     #tmpDBRecipe;
      L     DIW 104;	// ParNrOfIngrPerRecipe
      T     #tmpNrOfIngr;
      L     DIW 106;	// SCDB.ParNrOfByPerIngr
      SLD   3;
      T     #tmpNrOfBitIngr;
      L     DIW 32;	// CWA.ParDBBinControl
      T     "GCS7_ScaleControlDB".VarTemp[3];	// OutputFB69.VarDBBinControl
      T     #tmpBinControlDB;
      L     0;	// 
      ==I;	// 
      JC    cOUT;	// -->NoDBBin-Control
      L     DIW 104;	// SCDB.par_NoOfIngrPerRecipe
      L     DIW 106;	// SCDB.par_NoOfByPerIngr
      *I;	// 
      L     "GCS7_ScaleControlDB".VarTemp[2];	// Input.RecipeMemory
      *I;	// 
      L     DIW 100;	// ParDWNrFirstRecipe
      +D;	// 
      SLD   3;
      T     #tmpAddrIngr;	// -> Address recipe
// --- Begin Loop ingredient ------
      L     0;
cLOI: T     #tmpCntIngr;
      L     #tmpNrOfIngr;
      >=I;
      JC    cOUT;
      OPN   DI [#tmpDBRecipe];	//  
      L     0;	// 
      L     DIW [#tmpAddrIngr];	// Ingr[n].bin_nr
      ==I;	// End of recipe
      JC    cOUT;
      >=I;	// Discharge scale
      JC    cNXI;
      OPN   DB [#tmpBinControlDB];	// >>>CALL DB-BinControl
      T     DBW 20;	// VarBinNr
      CALL  "GCS7_BinCtrlSub" (
           CODE                     := 2);	//   Methode ReadBin
      A     DBX 39.0;	// Bin.ErrBinNotFound
      JC    cNXI;
      S     DBX 25.1;	// Bin.InfPreselected [1.3]
      A     DBX 24.5;	// Bin.InfLowLevel
      S     DBX 24.6;	// Bin.InfLevelMiddle [1.3]
      L     DBW 20;	// VarBinNr     [1.3]
      AN    DBX 24.5;	// Bin.InfLowLevel
      O     DB8.DBX 39.0;	// --> output.fault
      JC    cStr;	// [1.3]
      S     DB8.DBX 39.0;	// --> output.fault
      T     "GCS7_ScaleControlDB".VarTemp[4];	// Var_bin_nr   [1.3]
cStr: OPN   DB [#tmpBinControlDB];	// >>>CALL DB-BinControl
      CALL  "GCS7_BinCtrlSub" (
           CODE                     := 3);	//   Methode StoreBin [1.3]
cNXI: L     #tmpAddrIngr;	// (increment read address)
      L     #tmpNrOfBitIngr;
      +D;
      T     #tmpAddrIngr;
      L     #tmpCntIngr;
      +     1;
      JU    cLOI;
// --- end loop ingredient------
cOUT: BEU;
cEND: NOP   0;
END_FUNCTION

FUNCTION "GCS7_LogConvert_10" : VOID	// FC 73
TITLE = LOG: Message Converter for LOG Entry Format 10
//COPYRIGHT:     (C) 2003 BY  BUEHLER LTD. 
//                            CH-9240 UZWIL  SWITZERLAND
//
//PRODUCT:      GCS7 
//
//TITLE:        Message Converter for LOG Entry Format 10
//
//--------------------------------------------------------------------------
//
//IDENT:        AUTOR:              DEPT:                       DATE:
//
//FC73.1.0      A. Egli             CT3                         08.12.2003
//              1st Release
//
//--------------------------------------------------------------------------
//
//PURPOSE:       DATA-CONVERT FOR PRINTER PER LOG WITH PC
//
//RESTRICTIONS:  S7
//
//--------------------------------------------------------------------------
//
AUTHOR : EA
FAMILY : GCS7LL
NAME : MECONV
VERSION : 1.0
VAR_INPUT
  ObjectNo : INT ;	//Is used for communication with PC
  MsgType : INT ;	//Is used for message translation
  ClassMsgTxt : WORD ;	//Contains MessageClass and MessageTextNumber
  OType : INT ;	//Object Type
  MsgFormat : INT ;
  OldValue : DINT ;	//Old Value to Report
  NewValue : DINT ;	//New Value to Report
END_VAR
VAR_TEMP
  tmpHeader : WORD ;
  tmpPara2 : WORD ;
  tmpObjectNo : WORD ;
  tmpLineNo : WORD ;
  tmpMsgType : WORD ;
  tmpGr : INT ;
  tmpIndex : INT ;
  tmpPara5 : WORD ;
  tmpPara6 : WORD ;
  tmpPara7 : WORD ;
  tmpPara8 : WORD ;
END_VAR
BEGIN
NETWORK
TITLE =  MESSAGE
//Standard GCS90
      L     #ObjectNo;	// Change type INT --> WORD
      T     #tmpObjectNo;
      L     #ClassMsgTxt;	// Load: HighByte= Class ¦ Low Byte= TextNo (8 Bit)
      SRW   8;	// Delete TextNo
      SLW   5;
      L     #MsgFormat;
      +I;	// add MessageFormatNo
      T     #tmpHeader;	//-> Header=Format := Class ¦ MsgFormatNo
      L     #ClassMsgTxt;	// Load: HighByte= Class ¦ Low Byte= TextNo (8 Bit)
      L     2#11111111;	// Delete Class
      AW;
      L     #MsgType;
      SLW   8;
      OW;
      T     #tmpPara2;	//-->Para2 := MsgType ¦ TextNo
      L     #OldValue;
      T     #tmpPara6;
      SRD   16;
      T     #tmpPara5;
      L     #NewValue;
      T     #tmpPara8;
      SRD   16;
      T     #tmpPara7;
      L     "GCS7_Gr_OutLine";
      T     #tmpLineNo;
      L     #MsgType;
      T     #tmpMsgType;
      A     "GCS7_Gr_OutLogOff";
      JC    EQ00;
      CALL  "SYS_LOG_EntryQueue" (
           DBNumber                 := 5,
           Header                   := #tmpHeader,
           Para1                    := #tmpObjectNo,
           Para2                    := #tmpPara2,
           Para3                    := #tmpLineNo,
           Para4                    := #tmpMsgType,
           Para5                    := #tmpPara5,
           Para6                    := #tmpPara6,
           Para7                    := #tmpPara7,
           Para8                    := #tmpPara8,
           Para9                    := W#16#0,
           Para10                   := W#16#0,
           Para11                   := W#16#0);	//---Call Message Entry--- /  Queue DB Number                 /  Format /  ObjectNumber /  MsgType ¦ TextNo /  Line /  MsgType S7 /  Old Value  /  Old Value /  New Value  /  New Value  /  not used  /  not used  /  not used
EQ00: NOP   0;
NETWORK
TITLE = End of Block
END_FUNCTION

FUNCTION "SYS_DPDiagMain" : VOID	// FC 75
TITLE = DP-Diagnisys Main
//COPYRIGHT:     (C) 2001 BY  BUEHLER LTD. 
//                            CH-9240 UZWIL  SWITZERLAND
//
//PRODUCT:       DP-Diagnosis
//
//TITLE:         DP-DiagMain
//
//-------------------------------------------------------------------------
//
//IDENT:        AUTOR:              DEPT:                         DATE:
//
//FC75.1A       K. Tischer          CT3                          28-MAY-2001
//              1st Release
//
//-------------------------------------------------------------------------
//
//PURPOSE:  - each mastersystem is a separate Network
//              - initial same Bit
//              - Call DP-Diagnostic (orig. Siemens) 
//              - Call additional Diagnostic for not Siemens Slaves
//              - reset same parameters
//
//RESTRICTIONS:   NEEDS SIEMENS FB76 (original FB125)
//                NEEDS FC76 additional Diagnostic for not Siemens Slaves
//
//Paramters to set:
//              - FB76 DP_Mastersystem (prepaired 1 .. 4)
//              - FB76 EXTERNAL_DP_INTERFACE 
//                     prepaired MASTERSYSTEM 1   : FALSE
//                               MASTERSYSTEM 2..4: TRUE
//
//-------------------------------------------------------------------------
//
//
AUTHOR : TiK
FAMILY : DP
NAME : DPDiagM
VERSION : 1.0
VAR_TEMP
  Single_Step_Slave : BOOL ;
  Single_Step_Error : BOOL ;
  Reset : BOOL ;
  Single_Diag : BOOL ;
  Sum_Slave_Diag_Int : BYTE ;	//Anzahl Slave Diagnosen
  DiagNo : BYTE ;	//tik
  ByteSrc : INT ;	//TIK
  Diag_Dat_Norm_Act : ARRAY  [0 .. 7 ] OF //tik
  BYTE ;
  Fault : BOOL ;	//tik
END_VAR
BEGIN
NETWORK
TITLE =
NETWORK
TITLE = Mastersystem 1
//dignostic DB: DB75
//
// Save PCC parameters
      A     DB75.DBX 2.2;
      S     #Single_Step_Slave;
      A     DBX 2.3;
      S     #Single_Step_Error;
      A     DBX 2.4;
      S     #Reset;
      A     DBX 2.5;
      S     #Single_Diag;
// Call DPDiagnostic (orig. Siemens)
      CALL  "SYS_DP-Diagnosis" , "SYS_DPInfoM1" (
           DIW 0                    := 1,
           DIX 2.0                  := FALSE);
      OPN   "SYS_DPInfoM1";
      CALL  "SYS_DPDiag1";
      A     DB75.DBX 2.2;
      A     #Single_Step_Slave;
      R     DBX 2.2;
      R     #Single_Step_Slave;
      A     DBX 2.3;
      A     #Single_Step_Error;
      R     DBX 2.3;
      R     #Single_Step_Error;
      A     DBX 2.4;
      A     #Reset;
      R     DBX 2.4;
      R     #Reset;
      A     DBX 2.5;
      A     #Single_Diag;
      R     DBX 2.5;
      R     #Single_Diag;
//Call Diagnostic not Siemens
//reset PCC parameters
NETWORK
TITLE = Mastersystem 2
//dignostic DB: DB76
// Save PCC parameters
      A     DB76.DBX 2.2;
      S     #Single_Step_Slave;
      A     DBX 2.3;
      S     #Single_Step_Error;
      A     DBX 2.4;
      S     #Reset;
      A     DBX 2.5;
      S     #Single_Diag;
      CALL  "SYS_DP-Diagnosis" , "SYS_DPInfoM2" (
           DIW 0                    := 2,
           DIX 2.0                  := TRUE);
      OPN   "SYS_DPInfoM2";
      CALL  "SYS_DPDiag1";
      A     DB76.DBX 2.2;
      A     #Single_Step_Slave;
      R     DBX 2.2;
      R     #Single_Step_Slave;
      A     DBX 2.3;
      A     #Single_Step_Error;
      R     DBX 2.3;
      R     #Single_Step_Error;
      A     DBX 2.4;
      A     #Reset;
      R     DBX 2.4;
      R     #Reset;
      A     DBX 2.5;
      A     #Single_Diag;
      R     DBX 2.5;
      R     #Single_Diag;
//Call Diagnostic not Siemens
//reset PCC parameters
NETWORK
TITLE = Mastersystem 3
//dignostic DB: DB77
// Save PCC parameters
      A     DB77.DBX 2.2;
      S     #Single_Step_Slave;
      A     DBX 2.3;
      S     #Single_Step_Error;
      A     DBX 2.4;
      S     #Reset;
      A     DBX 2.5;
      S     #Single_Diag;
      CALL  "SYS_DP-Diagnosis" , "SYS_DPInfoM3" (
           DIW 0                    := 3,
           DIX 2.0                  := TRUE);
      OPN   "SYS_DPInfoM3";
      CALL  "SYS_DPDiag1";
      A     DB77.DBX 2.2;
      A     #Single_Step_Slave;
      R     DBX 2.2;
      R     #Single_Step_Slave;
      A     DBX 2.3;
      A     #Single_Step_Error;
      R     DBX 2.3;
      R     #Single_Step_Error;
      A     DBX 2.4;
      A     #Reset;
      R     DBX 2.4;
      R     #Reset;
      A     DBX 2.5;
      A     #Single_Diag;
      R     DBX 2.5;
      R     #Single_Diag;
//Call Diagnostic not Siemens
//reset PCC parameters
NETWORK
TITLE = Mastersystem 4
//dignostic DB: DB78
// Save PCC parameters
      A     DB78.DBX 2.2;
      S     #Single_Step_Slave;
      A     DBX 2.3;
      S     #Single_Step_Error;
      A     DBX 2.4;
      S     #Reset;
      A     DBX 2.5;
      S     #Single_Diag;
      CALL  "SYS_DP-Diagnosis" , "SYS_DPInfoM4" (
           DIW 0                    := 4,
           DIX 2.0                  := FALSE);
      OPN   "SYS_DPInfoM4";
      CALL  "SYS_DPDiag1";
      A     DB78.DBX 2.2;
      A     #Single_Step_Slave;
      R     DBX 2.2;
      R     #Single_Step_Slave;
      A     DBX 2.3;
      A     #Single_Step_Error;
      R     DBX 2.3;
      R     #Single_Step_Error;
      A     DBX 2.4;
      A     #Reset;
      R     DBX 2.4;
      R     #Reset;
      A     DBX 2.5;
      A     #Single_Diag;
      R     DBX 2.5;
      R     #Single_Diag;
//Call Diagnostic not Siemens
//reset PCC parameters
END_FUNCTION

FUNCTION "SYS_DPDiag1" : VOID	// FC 76
TITLE = DP-additional Diag
//COPYRIGHT:     (C) 2001 BY  BUEHLER LTD. 
//                            CH-9240 UZWIL  SWITZERLAND
//
//PRODUCT:       DP-Diagnosis
//
//TITLE:         DP-additional Diag
//
//-------------------------------------------------------------------------
//
//IDENT:        AUTOR:              DEPT:                         DATE:
//
//FC76.1B       K. Tischer          CT3                          20-Febr-2003
//              new buskoppler Wago 750-333 added
//FC76.1A       K. Tischer          CT3                          28-MAY-2001
//              1st Release
//
//-------------------------------------------------------------------------
//
//PURPOSE:  - each mastersystem is a separate Network
//              - initial same Bit
//              - Call DP-Diagnostic (orig. Siemens) 
//              - Call additional Diagnostic for not Siemens Slaves
//              - reset same parameters
//
//RESTRICTIONS:   NEEDS SIEMENS FB76 (original FB125)
//                NEEDS FC75 Main Diagnostic
//
//
//-------------------------------------------------------------------------
//
//
AUTHOR : TiK
FAMILY : DP
NAME : DPDiag1
VERSION : 1.0
VAR_TEMP
  Sum_Slave_Diag_Int : BYTE ;	//summary Slave Diagnosen
  ErrorNo : BYTE ;	//TiK
  ByteStart : INT ;	//TiK
  Diag_Lentgh : BYTE ;	//TiK
  Adr : DINT ;	//adress1
  Adr2 : DINT ;	//Adress 2
END_VAR
BEGIN
NETWORK
TITLE = check is diagtic present
      AN    DBX 932.3;	// additional diagnostic data present
      BEC;
NETWORK
TITLE = WAxx Wago (B750) 
//additianal Diagnisis for Wago Slaves Type (B750)
//
// - check result from SIEMENS FB76 => error type = device diagnosis
// - check result from SIEMENS FB76 => slave ident = B750
//
      NOP   0;
// error type = device diagnosis
      A(;
      L     DBB 11;	// error typ
      L     5;	// check device diagnostic
      ==I;
      );
// slave ident = B750
      A(;
      L     DBW 8;	// slave ident
      L     W#16#B750;	// B750 = Wago
      ==I;
      );
      JCN   WA00;	// jump end
// Init wago standard
      L     8;	// standard length of wago diagnostic data
      T     #Diag_Lentgh;
      L     DBB 1398;	// old error no (stored)
      T     #ErrorNo;	// error no
// calc summary DiagData
      L     DBB 938;	// norm diag data byte 6 (length)
      +     -2;	// 2 byte length info
      L     #Diag_Lentgh;	// Wago standard length =8
      /I;
      T     #Sum_Slave_Diag_Int;	// summary diag data
// Diag counter intialisieren
      A     DBX 2.3;	// single step error
      JCN   WA07;
// Diag counter inkrementieren
      L     #ErrorNo;	// actual diagnostic data no
      +     1;	// inkrement 1
      T     #ErrorNo;	// actual diagnostic data no
// Diag conter upper and lower limit
WA07: A(;
      L     #ErrorNo;
      L     #Sum_Slave_Diag_Int;	// upper limit 
      >I;
      );
      O(;
      L     #ErrorNo;
      L     1;	// lower limit
      <I;
      );
      JCN   WA06;
      L     1;	// set count diag =1
      T     #ErrorNo;	// out of range
WA06: NOP   0;
// write diagnostic to siemens DB
      L     #ErrorNo;
      T     DBB 10;	// => error number
      T     DBB 1398;	// => reserve byte siemens to store old error number
// calc start byte
      L     #ErrorNo;	// actual diagnostic data no
      L     #Diag_Lentgh;	// length diagnostic data
      *D;	// offset to start byte
      L     932;	// start byte diagnostic data
      +D;
      T     #ByteStart;	// => byte src diagnostic data
// ==check for Profibus or Klemmbus Diagnosis (first byte diagnostic data=0)===================      
      L     0;	// byte no
      L     #ByteStart;	// byte no start actual data
      +D;
      SLD   3;	// convert to bit value
      T     #Adr;	// store bit value
      L     DBB [#Adr];	// first byte diagnostic data
      L     0;
      ==I;
      JC    WA02;	//>>jump to check Klembus diagnosis >>>>>>>>>>>>>>>>>>>
// Modul / Kanal Diagnose ============================
      L     DBB [#Adr];	// first byte diagnostic data
      T     DBB 12;	// => modul no
      L     1;	// byte no
      L     #ByteStart;	// byte no start actual data
      +D;
      SLD   3;	// convert to bit value
      T     #Adr;	// store bit value
      L     DBB [#Adr];
      T     DBB 14;	// => cannel no
// Error analyse
      L     4;	// byte no
      L     #ByteStart;	// byte no start actual data
      +D;
      SLD   3;	// convert to bit value
      T     #Adr;	// store bit value
// == check Lower limit violated ======
      L     DBB [#Adr];
      L     2#100000001;	// compare bit 0 set
      AW;
      L     0;
      JCN   WA05;	// >> jump to check overrange >>>>>>>>>>>>>>>>>>>>>>>>>
      L     8;	//  8=Lower limit violated
      JU    WA03;	// >> jump to => canal error code >>>>>>>>>>>>>>>>>>>>>
// == check Upper limit violated ======
WA05: L     DBB [#Adr];
      L     2#100000010;	// compare bit 1 set
      AW;
      JCN   WA04;	// >> jump to other fault
      L     7;	// 7=Upper limit violated
      JU    WA03;	// >> jump to => canal error code >>>>>>>>>>>>>>>>>>>>>
WA04: L     DBB [#Adr];
      L     2#101000000;	// compare bit 6 set
      AW;
      JCN   WA03;	// >> jump to => canal error code >>>>>>>>>>>>>>>>>>>>>
      L     9;	// 9= Fault (e.g. encoder supply, load voltage at the output...;
WA03: T     DBW 16;	// => canal error code
      L     3;	// 3= channel error
      T     DBB 11;	// => error type
      JU    WA00;	// jump end
WA02: NOP   0;	// << check Klemmbus diagnosis <<<<<<<<<<<<<<<<<<<<<<<<<
      L     1;	// byte no
      L     #ByteStart;	// byte no start actual data
      +D;
      SLD   3;	// convert to bit value
      T     #Adr;	// store bit value
      L     DBB [#Adr];
      L     0;
      ==I;
      JC    WA01;	//>>jump to Klemmbus diagnosis >>>>>>>>>>>>>>>>>>>>>>>>>
// Profibus Diagnosis =================================
      L     4;	// byte no
      L     #ByteStart;	// byte no start actual data
      +D;
      SLD   3;	// convert to bit value
      T     #Adr;	// store bit value
      L     DBB [#Adr];
      L     100;	// 100=not enough configuration data;200=error in 1st configuration byte;300=non-supported module at position N
      *I;
      T     DBB 13;	// => modul state
      L     2;	// 2=Modul Diagnosis
      T     DBB 11;	// => error type
      JU    WA00;	// >> jump end >>>>>>>>>>>>>>>>>>>>>>>>>>>>>>>>>>>>>>>>>>>
// << Klemmenbus Diagnosis <<<<<<<<<<<<<<<<<<<<<<<<<<<<<<<
WA01: NOP   0;
// prepair modul no
      L     5;	// byte no
      L     #ByteStart;	// byte no start actual data
      +D;
      SLD   3;	// convert to bit value
      T     #Adr;	// store bit value
      L     DBB [#Adr];
      T     DBB 12;	// => modul no
// prepair modul state
      L     4;	// byte no
      L     #ByteStart;	// byte no start actual data
      +D;
      SLD   3;	// convert to bit value
      T     #Adr;	// store bit value
      L     DBB [#Adr];
      L     10;	// 10=EEPROM Checksum Error;20=error in programmed process image;30=modules have identified error in fieldbus commands;40=fieldbus break after module N
      *I;	// 50=filedbus error in register communication with module N;60=error in PROFIBUS-DP configuration telegram;70=non-supported module at position N
      T     DBB 13;	// => modul state
// prepair error type
      L     2;	// 2=Modul Diagnosis
      T     DBB 11;	// => error type
      JU    WA00;	// jump end
WA00: NOP   0;
NETWORK
TITLE = WAxx Wago (B754) 
//additianal Diagnisis for Wago Slaves Type (B750-333)
//
// - check result from SIEMENS FB76 => error type = device diagnosis
// - check result from SIEMENS FB76 => slave ident = B750
//
      NOP   0;
// error type = device diagnosis
      A(;
      L     DBB 11;	// error typ
      L     5;	// check device diagnostic
      ==I;
      );
// slave ident = B750-333
      A(;
      L     DBW 8;	// slave ident
      L     W#16#B754;	// B754 = Wago
      ==I;
      );
      JCN   WB00;	// jump end
// Init wago standard
      L     3;
      T     #Diag_Lentgh;	// kanaldiagsostic standard length =3
      L     DBB 1398;	// old error no (stored)
      T     #ErrorNo;	// error no
// calc summary DiagData
      L     DBB 44;	// length of diagnostic data (SFC13) incl. header
      L     22;	// 22 byte (header=6Byte; kennungdata=9Byte; modulstate=7
      >=I;
      JCN   WB00;
      L     DBB 44;	// length of diagnostic data (SFC13) incl. header
      +     -22;	// 22 byte (header=6Byte; kennungdata=9Byte; modulstate=7
      L     3;	// Wago standard length =3
      /I;
      T     #Sum_Slave_Diag_Int;	// summary diag data
// Diag counter intialisieren
      A     DBX 2.3;	// single step error
      JCN   WB07;
// Diag counter inkrementieren
      L     #ErrorNo;	// actual diagnostic data no
      +     1;	// inkrement 1
      T     #ErrorNo;	// actual diagnostic data no
// Diag conter upper and lower limit
WB07: A(;
      L     #ErrorNo;
      L     #Sum_Slave_Diag_Int;	// upper limit 
      >I;
      );
      O(;
      L     #ErrorNo;
      L     1;	// lower limit
      <I;
      );
      JCN   WB06;
      L     1;	// set error no =1
      T     #ErrorNo;	// out of range
WB06: NOP   0;
// write diagnostic to siemens DB
      L     #ErrorNo;
      T     DBB 10;	// => error number
      T     DBB 1398;	// => reserve byte siemens to store old error number
// ==check for Profibus or Klemmbus Diagnosis (first byte diagnostic data=0)===================      
      L     951;	//byte 20 => device diagnostic 
      SLD   3;
      T     #Adr;
      L     952;
      SLD   3;
      T     #Adr2;
      L     DBB [#Adr];	// state message 0= no error
      L     0;
      >I;
      JCN   WB10;
      L     2;	// 2=Modul Diagnosis
      T     DBB 11;	// => error type
      L     DBB [#Adr2];
      T     DBB 12;	// => modul no
      L     DBB [#Adr];
      T     DBB 13;	// => modul state
      L     0;
      T     DBW 16;	// => error no
      JU    WB00;	// >> jump end >>>>>>>>>>>>>>>>>>>>>>>>>>>>>>>>>>>>>>>>>>>
// << Klemmenbus Diagnosis <<<<<<<<<<<<<<<<<<<<<<<<<<<<<<<
WB10: NOP   0;
// calc start byte
      L     #ErrorNo;	// actual diagnostic data no
      L     #Diag_Lentgh;	// length diagnostic data (3Byte)
      *D;	// offset to start byte
      L     951;	// start byte diagnostic data
      +D;
      T     #ByteStart;	// => byte src diagnostic data
// Kanal Diagnose ============================
      L     3;	// 3= channel error
      T     DBB 11;	// => error type
      L     #ByteStart;
      SLD   3;
      T     #Adr;
      L     DBB [#Adr];	// first byte diagnostic data
      L     B#16#3F;
      AW;
      T     DBB 12;	// => modul no
      L     1;	// byte no
      L     #ByteStart;	// byte no start actual data
      +D;
      SLD   3;	// convert to bit value
      T     #Adr;	// store bit value
      L     DBB [#Adr];
      L     B#16#3F;
      AW;
      T     DBB 14;	// => cannel no
      L     2;	// byte no
      L     #ByteStart;	// byte no start actual data
      +D;
      SLD   3;	// convert to bit value
      T     #Adr;	// store bit value
      L     DBB [#Adr];
      L     B#16#1F;
      AW;
      T     DBW 16;	// => error no
WB00: NOP   0;
END_FUNCTION

FUNCTION "GCS7BinCtrlUpdataLevel" : VOID	// FC 78
TITLE = BinMain
//COPYRIGHT:    (C) 1994 BY  BUHLER LTD.
//                           CH-9240 UZWIL  SWITZERLAND
//
//PRODUCT:      GCS7
//
//TITLE:        BIN CONTROL: Update Bin Level
// 
//-------------------------------------------------------------------------
//
//IDENT:        AUTOR:              DEPT:                         DATE:
//FC78.1.5       A.Egli              CT3                           07-Jul-2004
//               Binlist InDPFaultLL, InDPFaultHL
//FC78.1.4       A.Egli              CT3                           20-Apr-2004
//               Send Override only to active bin
//FC78.1.3       A.Egli              CT3                           26-Mar-2004
//               When StaSameSndRcv: Do not add Overfillweight
//FC78.1.2       A.Egli              CT3                           03-Nov-2003
//               "BinDB".PCRead.Status.StaSameSndRcv
//FC78.1.1       K.Tischer           CT3                           27-Oct-2003
//               set CmdLastReceiverActive only for activ bin
//FC78.1.0       A.Egli              CT3                           07-Oct-2002
//               New release 
//
//-------------------------------------------------------------------------
//
//PURPOSE:      MANUAL : BINMAN
//              Communication between Bin list and Centtal Bin List 
//
//RESTRICTIONS:
//
//-------------------------------------------------------------------------
//
//ACTUAL DB BY CALL: DB Bin control
//
//-------------------------------------------
//Input Parameter:
//----------------
//MODE
//   0 : With overfilling
//       Sender list    : Bin(x).InfLevelFault :=OutLowLevel
//       Reveiver list  : Bin(x).InfLevelFault :=OutHighLevel
//   1 : No overfilling (used for mixing line)
//       Sender list    : Bin(x).InfLevelFault :=InLowLevel
//       Reveiver list  : Bin(x).InfLevelFault :=InHighLevel
//
//Flowrate: 
//    Actual flowrate kg/h
//    With this flowrate the weight "InOutFillingWeight" and 
//    "InOutOverFillingWeight" are counting.
//
//-------------------------------------------
//Output Parameter:
//----------------
//
//-------------------------------------------
//Global Output Data:
//------------------
//// "BinDB".Bin(x).InfLowLevel
//// "BinDB".Bin(x).InfHighLevel
//// "BinDB".Bin(x).InfLevelFault
//// "BinDB".Bin(x).InfFeedOff
//// "PLC_BinListDB".Bin(x).CmdFilling
//// "PLC_BinListDB".Bin(x).CmdDischarging
//// "PLC_BinListDB".Bin(x).CmdOverrideHL
//// "PLC_BinListDB".Bin(x).CmdOverrideLL
//// "PLC_BinListDB".Bin(x).InReceiverCounter
//
//
AUTHOR : EA
FAMILY : GCS7UL
NAME : BIN_MAN2
VERSION : 1.5
VAR_INPUT
  MODE : INT ;	//CODE
  Flowrate : DINT ;	//kg/h
END_VAR
VAR_TEMP
  varBinDB : INT ;
  VarAddrBin : DWORD ;
  VarAddrBinIdx : DWORD ;
  VarAddrIdx : DWORD ;
  VarCnt : INT ;
  VarLenBinBit : DINT ;
  VarIngrIdx : INT ;
  VarCntBin : INT ;
  VarBinNr : INT ;
  VarCentBinIdx : INT ;
  VarAddrCentBin : DWORD ;
  VarCentLenBinBit : DINT ;
  tmpFlowrateKgS : REAL ;	//[kg/s]
  tmpMode_1_No : BOOL ;	//No overfilling
END_VAR
BEGIN
NETWORK
TITLE =
      L     DBNO;
      T     #varBinDB;
      OPN   DI [#varBinDB];
      L     DBW 10;	// "BinDB".Para.ParNoOfBytePerBin
      SLD   3;
      T     #VarLenBinBit;
//Mode: No overfilling
      L     #MODE;
      L     1;
      ==I;
      =     #tmpMode_1_No;
NETWORK
TITLE = Calulate Florate per second
      L     0.000000e+00;
      AN    "SYS_Tick1s";
      JC    C1;
      L     #Flowrate;	// [kg/h]
      DTR;
      L     3.600000e+03;
      /R;
C1:   T     #tmpFlowrateKgS;	//[kg/s]
NETWORK
TITLE =  Length Test
      L     DBW 10;	// "BinDB".Para.ParNoOfBytePerBin
      L     DBW 12;	// "BinDB".Para.ParNoOfBin
      *I;
      L     DBW 8;	// "BinDB".Para.ParByteFirstBin
      +I;
      L     DBLG;	//  Actual DB Lenght
      >I;
      JCN   aEnd;
      BEU;
aEnd: NOP   0;
NETWORK
TITLE = Update Bin
//Start Adress Loop
      L     DIW 8;	//"BinDB".Para.ParByteFirstBin
      SLD   3;
      T     #VarAddrBin;	//--> Pointer to Bin
//--loop bin -------------------------------------------
      L     0;
      L     DIW 12;	//  "BinDB".Para.ParNoOfBin
      ==I;
      BEC;
uLop: T     #VarCntBin;	// var_loop_bin_counter
      L     #VarAddrBin;
      L     #VarLenBinBit;
      +D;
      +     L#-16;
      T     #VarAddrBinIdx;	//   
      LAR1  #VarAddrBin;
      L     DIW [AR1,P#0.0];
      T     #VarBinNr;
      L     DIW [AR1,P#2.0];	// binlist[n].Bin status word
      T     DIW 24;	// ->var_bin_status
      L     DIW [#VarAddrBinIdx];	// binlist[n].Bin status word
      T     #VarCentBinIdx;	//Index of bin in Central Bin List
//Search bin in Central Bin List
      L     "PLC_BinListDB".Para.ParNoOfBytePerBin;
      SLD   3;
      T     #VarCentLenBinBit;
//Calculate old address in central bin lsit
      L     #VarCentBinIdx;	//Index of bin in Central Bin List
      +     -1;
      L     "PLC_BinListDB".Para.ParNoOfBytePerBin;
      *I;
      L     "PLC_BinListDB".Para.ParByteFirstBin;
      +I;
      SLD   3;
      T     #VarAddrCentBin;
//Check Index
      L     1;
      L     #VarCentBinIdx;	//Index of bin in Central Bin List
      >I;
      JC    USEA;
      L     "PLC_BinListDB".Para.ParNoOfBin;
      >I;
      JC    USEA;
//Check old bin number
      LAR2  #VarAddrCentBin;
      L     DBW [AR2,P#0.0];	//PLC_BinListDB".BinXxx.ParBinNr
      L     #VarBinNr;
      ==I;
      JC    UOK;
//================================================
//Search position because Bin has moved
USEA: L     "PLC_BinListDB".Para.ParByteFirstBin;
      SLD   3;
      T     #VarAddrCentBin;
      L     1;
UZLo: T     #VarCentBinIdx;
      L     "PLC_BinListDB".Para.ParNoOfBin;
      >I;
      JC    UErr;
      L     DBW [#VarAddrCentBin];	//PLC_BinListDB".BinXxx.ParBinNr
      L     #VarBinNr;
      ==I;
      JC    UFND;	//--> Found
      L     #VarAddrCentBin;
      L     #VarCentLenBinBit;
      +D;
      T     #VarAddrCentBin;	//   
      L     #VarCentBinIdx;
      +     1;
      JU    UZLo;	//End of Loop Cental Bin List
//================================================
//Error Bin not found
UErr: L     0;	//Index of bin in Central Bin List
      T     #VarAddrBinIdx;
      S     DIX 24.2;	//"BinDB".VarTemp.Bin.InFeedOff
      JU    uSAV;
//Store Index if bin found
UFND: LAR1  #VarAddrBinIdx;
      L     #VarCentBinIdx;	//Index of bin in Central Bin List
      T     DIW [AR1,P#0.0];	// binlist[n].Bin status word
//================================================
//Update
UOK:  LAR2  #VarAddrCentBin;
// --------------------------------------------------
// Copy data of actual Bin to "PLC_BinListDB".tmpBin
      L     DBD [AR2,P#2.0];
      T     DB79.DBD 22;
      L     DBD [AR2,P#6.0];
      T     DB79.DBD 26;
      L     DBD [AR2,P#10.0];
      T     DB79.DBD 30;
      L     DBD [AR2,P#14.0];
      T     DB79.DBD 34;
//----------------------------------------
//Receiver List
//----------------------------------------
      A     DIX 7.2;	//"BinDB".Para.ParTypeDef.ParSenderList
      JC    USD;
// Check List used
      A     DIX 105.5;	//"BinDB".PCRead.Status.StaListNotUsed
      JC    URC3;
// Send Command CmdLastReceiverActive                                            [1.1]
      A     DIX 25.0;	//"BinDB".VarTemp.Bin.InfActiveBin       [1.1]
      AN    DIX 25.2;	//"BinDB".VarTemp.Bin.InfDeselect        [1.1]
      A     DIX 104.0;	//"BinDB".PCRead.Status.StaLastBinActive [1.1]
      S     "PLC_BinListDB".tmpBin.CmdLastReceiverActive;	//                   [1.1]
// Send Command CmdFilling
      A     DIX 25.0;	//"BinDB".VarTemp.Bin.InfActiveBin
      A     DIX 104.1;	//"BinDB".PCRead.Status.StaFeeding
      S     "PLC_BinListDB".tmpBin.CmdFilling;
      JCN   URC2;
// Counter active receiver
      L     "PLC_BinListDB".tmpBin.InReceiverCounter;
      +     1;
      T     "PLC_BinListDB".tmpBin.InReceiverCounter;
// Add FillingWeight
      L     "PLC_BinListDB".tmpBin.InOutFillingWeight;
      L     #tmpFlowrateKgS;
      +R;
      JO    URC1;
      T     "PLC_BinListDB".tmpBin.InOutFillingWeight;
// Add OverfillWeight
URC1: AN    "PLC_BinListDB".tmpBin.InHighLevel;
      O     DIX 105.4;	// "BinDB".PCRead.Status.StaSameSndRcv [1.3] 
      JC    URC2;
      L     "PLC_BinListDB".tmpBin.InOutOverfillWeight;
      L     #tmpFlowrateKgS;
      +R;
      JO    URC2;
      T     "PLC_BinListDB".tmpBin.InOutOverfillWeight;
// Send Command StaOverrideLevel
URC2: A     DIX 104.2;	//"BinDB".PCRead.Status.StaOverrideLevel
      AN    DIX 105.5;	//"BinDB".PCRead.Status.StaListNotUsed  [1.4]
      A     DIX 25.0;	//"BinDB".VarTemp.Bin.InfActiveBin [1.4]
      S     "PLC_BinListDB".tmpBin.CmdOverrideHL;
// Read InfLevelFault
URC3: A     "PLC_BinListDB".tmpBin.InHighLevel;
      A     #tmpMode_1_No;
      O     "PLC_BinListDB".tmpBin.OutHighLevel;
      AN    DIX 105.4;	// "BinDB".PCRead.Status.StaSameSndRcv [1.2]
      =     DIX 24.1;	// "BinDB".VarTemp.Bin.InfLevelFault
// Read InFeedOff
      A     "PLC_BinListDB".tmpBin.OutFull;
      A     DIX 25.0;	//"BinDB".VarTemp.Bin.InfActiveBin 
      O     "PLC_BinListDB".tmpBin.InFeedOffHL;
      AN    DIX 105.4;	// "BinDB".PCRead.Status.StaSameSndRcv [1.2]
      =     DIX 24.2;	//"BinDB".VarTemp.Bin.InFeedOff
// Read DryFillingDoone
      A     "PLC_BinListDB".tmpBin.OutDryFillingDone;
      =     DIX 24.3;	//"BinDB".VarTemp.Bin.OutDryFillingDone
// Read DPFault                                                             //[1.5]
      A     "PLC_BinListDB".tmpBin.InDPFaultHL;	//[1.5]
      =     DIX 25.4;	//"BinDB".VarTemp.Bin.InOutDPFault //[1.5]
      JU    UNXT;
//----------------------------------------
//Sender List
//----------------------------------------
// Send Command Discharging
USD:  A     DIX 25.0;	//"BinDB".VarTemp.Bin.InfActiveBin
      A     DIX 104.1;	//"BinDB".PCRead.Status.StaFeeding
      S     "PLC_BinListDB".tmpBin.CmdDischarging;
      JCN   USD3;
// Add FillingWeight
      L     "PLC_BinListDB".tmpBin.InOutFillingWeight;
      L     #tmpFlowrateKgS;
      -R;
      JP    USD2;
      L     0.000000e+00;
USD2: T     "PLC_BinListDB".tmpBin.InOutFillingWeight;
// Send Command StaOverrideLevel
USD3: AN    DIX 105.5;	//"BinDB".PCRead.Status.StaListNotUsed
      A     DIX 104.2;	//"BinDB".PCRead.Status.StaOverrideLevel
      A     DIX 25.0;	//"BinDB".VarTemp.Bin.InfActiveBin [1.4]
      S     "PLC_BinListDB".tmpBin.CmdOverrideLL;
// Read InfLevelFault
      A     "PLC_BinListDB".tmpBin.InLowLevel;
      A     #tmpMode_1_No;
      O     "PLC_BinListDB".tmpBin.OutLowLevel;
      AN    DIX 105.4;	// "BinDB".PCRead.Status.StaSameSndRcv [1.2]
      =     DIX 24.1;	// "BinDB".VarTemp.Bin.InfLevelFault
// Read InFeedOff
      A     "PLC_BinListDB".tmpBin.InFeedOffLL;
      AN    DIX 105.4;	// "BinDB".PCRead.Status.StaSameSndRcv [1.2]
      =     DIX 24.2;	//"BinDB".VarTemp.Bin.InFeedOff
// Read DPFault                                                             //[1.5]
      A     "PLC_BinListDB".tmpBin.InDPFaultLL;	//[1.5]
      =     DIX 25.4;	//"BinDB".VarTemp.Bin.InOutDPFault //[1.5]
//Read HL und LL
UNXT: NOP   0;
      A     "PLC_BinListDB".tmpBin.InLowLevel;
      =     DIX 24.5;	// bin[n]."BinDB".VarTemp.Bin.InfLowLevel
      A     "PLC_BinListDB".tmpBin.InHighLevel;
      =     DIX 24.7;	// bin[n]."BinDB".VarTemp.Bin.InfHighLevel
// --------------------------------------------------
// Store Data 
// --------------------------------------------------
// Copy data of "PLC_BinListDB".tmpBin back to list
      LAR2  #VarAddrCentBin;
      L     DB79.DBD 22;
      T     DBD [AR2,P#2.0];
      L     DB79.DBD 26;
      T     DBD [AR2,P#6.0];
      L     DB79.DBD 30;
      T     DBD [AR2,P#10.0];
      L     DB79.DBD 34;
      T     DBD [AR2,P#14.0];
//---------------------------------------------
//Store Bin
uSAV: LAR1  #VarAddrBin;
      L     DIW 24;	// ->var_bin_status
      T     DIW [AR1,P#2.0];	// binlist[n].Bin status word
      L     #VarCentBinIdx;	//Index of bin in Central Bin List
      T     DIW [#VarAddrBinIdx];	// binlist[n].Bin status word
//---------------------------------------------
//Next Bin of actual list
      L     #VarAddrBin;
      L     #VarLenBinBit;
      +D;
      T     #VarAddrBin;
      L     #VarCntBin;
      LOOP  uLop;
      BEU;
      NOP   0;
END_FUNCTION

// FC 90: know-how protected block, not included

// FC 91: know-how protected block, not included

// FC 92: know-how protected block, not included

// FC 93: know-how protected block, not included

FUNCTION "SYS_SimpleDPInfo" : VOID	// FC 98
TITLE = Simple DP-Diagnostic
//
//COPYRIGHT:    (C) 1999 BY  BUHLER LTD.
//                           CH-9240 UZWIL  SWITZERLAND
//
//PRODUCT:      S7
//
//TITLE:        Simple DP-Diagnostic
//
//-------------------------------------------------------------------------
//
//IDENT:        AUTHOR:             DEPT:                       DATE:
//
//FC98.1A       S. Kalberer         CT3                         09.Aug.1999
//              1st Release in S7
//
//-------------------------------------------------------------------------
//
//PURPOSE:      MANUAL : see Siemens manual DIAG21_d.PDF
//RESTRICTIONS: S7 type: see also Siemens manual
//
//-------------------------------------------------------------------------
//Input Parameters:
//-----------------
//
// InEnableCheck: 
//                FALSE = DP-Diagnostic check inactive
//                TRUE  = DP-Diagnostic check active
// InExtDPInterface (only relevant for S7-400):
//                FALSE = S7-300/ Internal Master DP-Interface (Master-CPU)
//                TRUE  = External Master DP-Interface  (CP, IM)
// InDPMasterSystemNo:
//                Number of DP-Mastersystems that was projected with STEP 7
//                (1= standard)
//
AUTHOR : SK
FAMILY : DP
NAME : DP_Diag
VERSION : 1.0
VAR_INPUT
  InEnableCheck : BOOL ;	//Signal to enable the diagnostic check
  InExtDPInterface : BOOL ;	//only S7-400: 0= integrated (Master-CPU), 1= external (CP, IM)
  InDPMasterSystemNo : INT ;	//DP-Master System Number (prjected with STEP 7)
END_VAR
BEGIN
NETWORK
TITLE = Call Siemens FC 99 (GLOBAL_DP_INFO)
      CALL  "SIEMENS_GlobalDPInfo" (
           $1                       := #InEnableCheck,
           $2                       := #InExtDPInterface,
           $3                       := #InDPMasterSystemNo,
           $4                       := "SYS_SimpleDPInfo4DB".tmpDataField,
           $5                       := "SYS_SimpleDPInfo4DB".Sum_SlavesNotPresent,
           $6                       := "SYS_SimpleDPInfo4DB".List_SlavesNotPresent,
           $7                       := "SYS_SimpleDPInfo4DB".List_SlavesError,
           $8                       := "SYS_SimpleDPInfo4DB".OutRetVal,
           $9                       := "SYS_SimpleDPInfo4DB".OutBusy);
END_FUNCTION

// FC 99: know-how protected block, not included

FUNCTION "SYS_GeneralPLCStartup" : VOID	// FC 100
TITLE = General plc startup functions
//COPYRIGHT:      (C) 2000 BY  BUHLER LTD.
//                           CH-9240 UZWIL  SWITZERLAND
//
//PRODUCT:        PROEJCT
//
//TITLE:          General PLC startup functions
//
//                Generelle SPS-Anlauffunktionen
//
//
//--------------------------------------------------------------------------------
//
//IDENT:          AUTOR:            DEPT:                             DATE:
//
//P01_FC100.1.0   A.Egli            CT3                               14-Jul-2004
//                1st Release
//
//--------------------------------------------------------------------------------
//
//PURPOSE:      
//
//RESTRICTIONS: 
//
//--------------------------------------------------------------------------------
//
//
AUTHOR : EA
FAMILY : ASW
VERSION : 9.9
BEGIN
NETWORK
TITLE = End of block
      BE;
END_FUNCTION

FUNCTION "ConvertGrayCode" : VOID	// FC 108
TITLE = Convert Gray Code
//COPYRIGHT:    (C) 2003 BY  BUHLER AG
//                           CH-9240 UZWIL  SWITZERLAND
//
//PRODUCT:      GCS7
//
//TITLE:        Convert Gray Code Value to Integer
//              
//
//-------------------------------------------------------------------------
//
//IDENT:        AUTHOR:             DEPT:             DATE:
//
//FC109.1A      A.Egli              CT3               05-Apr-2003
//              1st Release
//
//-------------------------------------------------------------------------
//
//PURPOSE: 
//
//RESTRICTIONS: 
//
//-------------------------------------------------------------------------
//
//Code example for VB6.0
//======================
//
//Public Function IntToGary(ByVal aValue As Long) As Long
//Dim i As Integer
//Dim v As Long
//Dim out As Long
// v = aValue
// out = 0
// For i = 16 To 0 Step -1
//   If v >= bitValue(i) Then
//    out = out Or bitValue(i)
//    v = bitValue(i + 1) - v - 1
//   End If
// Next i
// IntToGary = out
//End Function
//
//Public Function GaryToInt(ByVal aValue As Long) As Long
//Dim i As Integer
//Dim v As Long
//Dim out As Long
// v = aValue
// out = 0
// For i = 0 To 16
//  'Test if bit is 1
//  If (v And bitValue(i)) <> 0 Then
//    out = bitValue(i + 1) - out - 1
//  End If
// Next i
// GaryToInt = out
//End Function
//
//
//
//
//
//
//
//
AUTHOR : GS
FAMILY : ASW
NAME : ANA_S5_S
VERSION : 1.0
VAR_INPUT
  GrayCode : WORD ;	//Value as Gray Code
END_VAR
VAR_OUTPUT
  OutValue : INT ;	//Value as Integer
END_VAR
VAR_TEMP
  tmpBitValue : DINT ;
  tmpValue : DINT ;
  tmpOutValue : DINT ;
END_VAR
BEGIN
NETWORK
TITLE = Initialisation
      L     0;
      T     #tmpOutValue;
      L     1;
      T     #tmpBitValue;
      L     #GrayCode;
      T     #tmpValue;
NETWORK
TITLE = Convert
LOP1: L     0;
      L     #tmpValue;
      ==D;
      JC    OUT;
      SRD   1;
      T     #tmpValue;
      JP    Is1;	//Jump when Bit is 1
      JU    NEXT;
//Calculate, if bit is 1
Is1:  L     #tmpBitValue;
      SLD   1;
      L     #tmpOutValue;
      -D;
      L     1;
      -D;
      T     #tmpOutValue;
//======================
NEXT: L     #tmpBitValue;
      SLD   1;
      T     #tmpBitValue;
      JU    LOP1;
OUT:  NOP   0;
NETWORK
TITLE =
      L     #tmpOutValue;
      T     #OutValue;
END_FUNCTION

